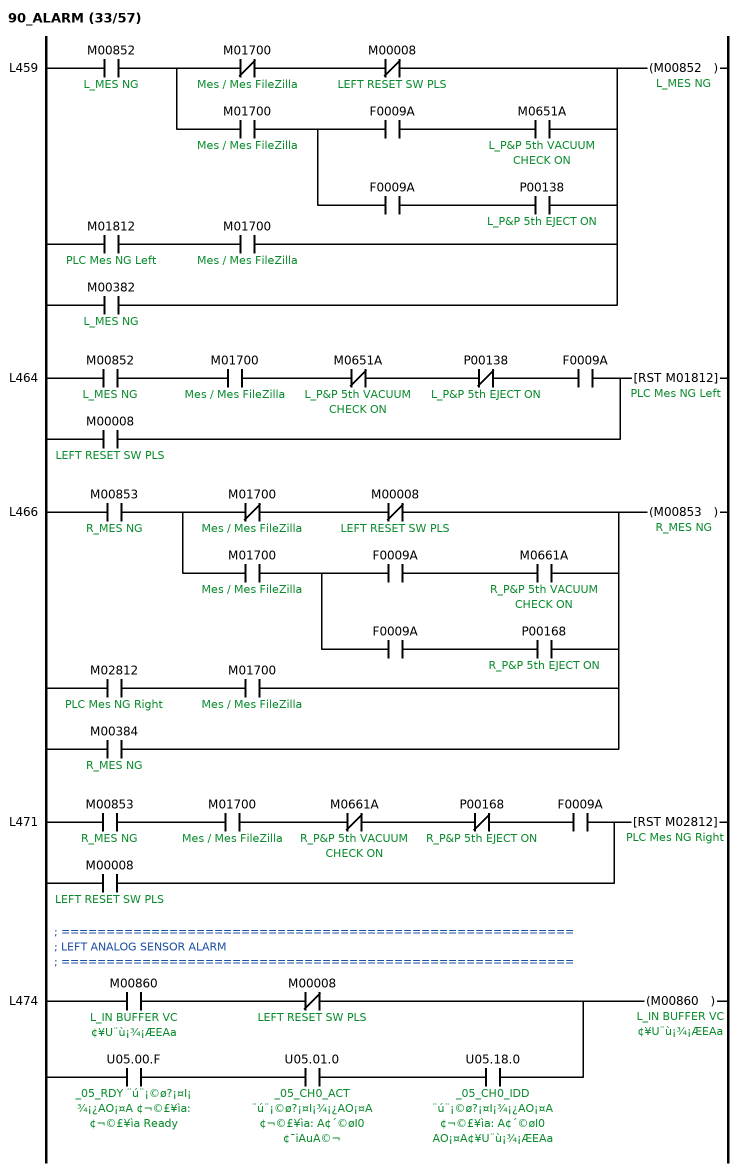
[picture p384: 90_ALARM rungs L459-L474]
; L459
LOAD      M00852	// L_MES NG
LOAD NOT  M01700	// Mes / Mes FileZilla
AND NOT   M00008	// LEFT RESET SW PLS
LOAD      M01700	// Mes / Mes FileZilla
LOAD      F0009A
AND       M0651A	// L_P&P 5th VACUUM CHECK ON
LOAD      F0009A
AND       P00138	// L_P&P 5th EJECT ON
OR LOAD
AND LOAD
OR LOAD
AND LOAD
LOAD      M01812	// PLC Mes NG Left
AND       M01700	// Mes / Mes FileZilla
OR LOAD
OR        M00382	// L_MES NG
OUT       M00852	// L_MES NG
; L464
LOAD      M00852	// L_MES NG
AND       M01700	// Mes / Mes FileZilla
AND NOT   M0651A	// L_P&P 5th VACUUM CHECK ON
AND NOT   P00138	// L_P&P 5th EJECT ON
AND       F0009A
OR        M00008	// LEFT RESET SW PLS
RST       M01812	// PLC Mes NG Left
; L466
LOAD      M00853	// R_MES NG
LOAD NOT  M01700	// Mes / Mes FileZilla
AND NOT   M00008	// LEFT RESET SW PLS
LOAD      M01700	// Mes / Mes FileZilla
LOAD      F0009A
AND       M0661A	// R_P&P 5th VACUUM CHECK ON
LOAD      F0009A
AND       P00168	// R_P&P 5th EJECT ON
OR LOAD
AND LOAD
OR LOAD
AND LOAD
LOAD      M02812	// PLC Mes NG Right
AND       M01700	// Mes / Mes FileZilla
OR LOAD
OR        M00384	// R_MES NG
OUT       M00853	// R_MES NG
; L471
LOAD      M00853	// R_MES NG
AND       M01700	// Mes / Mes FileZilla
AND NOT   M0661A	// R_P&P 5th VACUUM CHECK ON
AND NOT   P00168	// R_P&P 5th EJECT ON
AND       F0009A
OR        M00008	// LEFT RESET SW PLS
RST       M02812	// PLC Mes NG Right
// =========================================================
// 
//        LEFT ANALOG SENSOR ALARM
// 
// =========================================================
; L474
LOAD      M00860	// L_IN BUFFER VC ¢¥U¨ù¡¾¡ÆEAa
AND NOT   M00008	// LEFT RESET SW PLS
LOAD      U05.00.F	// _05_RDY ¨ú¨¡©ø?¡¤I¡¾¡¿AO¡¤A ¢¬©£¥ìa: ¢¬©£¥ìa Ready
AND       U05.01.0	// _05_CH0_ACT ¨ú¨¡©ø?¡¤I¡¾¡¿AO¡¤A ¢¬©£¥ìa: A¢´©øI0 ¢¯iAuA©¬
AND       U05.18.0	// _05_CH0_IDD ¨ú¨¡©ø?¡¤I¡¾¡¿AO¡¤A ¢¬©£¥ìa: A¢´©øI0 AO¡¤A¢¥U¨ù¡¾¡ÆEAa
OR LOAD
OUT       M00860	// L_IN BUFFER VC ¢¥U¨ù¡¾¡ÆEAa

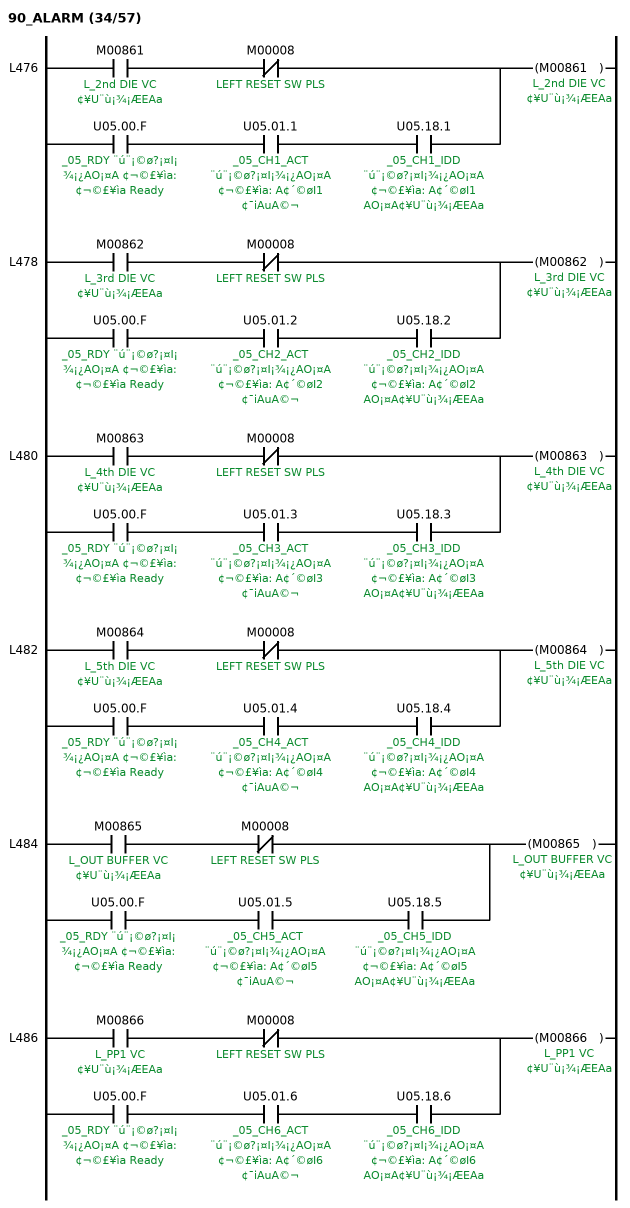
; L476
LOAD      M00861	// L_2nd DIE VC ¢¥U¨ù¡¾¡ÆEAa
AND NOT   M00008	// LEFT RESET SW PLS
LOAD      U05.00.F	// _05_RDY ¨ú¨¡©ø?¡¤I¡¾¡¿AO¡¤A ¢¬©£¥ìa: ¢¬©£¥ìa Ready
AND       U05.01.1	// _05_CH1_ACT ¨ú¨¡©ø?¡¤I¡¾¡¿AO¡¤A ¢¬©£¥ìa: A¢´©øI1 ¢¯iAuA©¬
AND       U05.18.1	// _05_CH1_IDD ¨ú¨¡©ø?¡¤I¡¾¡¿AO¡¤A ¢¬©£¥ìa: A¢´©øI1 AO¡¤A¢¥U¨ù¡¾¡ÆEAa
OR LOAD
OUT       M00861	// L_2nd DIE VC ¢¥U¨ù¡¾¡ÆEAa
; L478
LOAD      M00862	// L_3rd DIE VC ¢¥U¨ù¡¾¡ÆEAa
AND NOT   M00008	// LEFT RESET SW PLS
LOAD      U05.00.F	// _05_RDY ¨ú¨¡©ø?¡¤I¡¾¡¿AO¡¤A ¢¬©£¥ìa: ¢¬©£¥ìa Ready
AND       U05.01.2	// _05_CH2_ACT ¨ú¨¡©ø?¡¤I¡¾¡¿AO¡¤A ¢¬©£¥ìa: A¢´©øI2 ¢¯iAuA©¬
AND       U05.18.2	// _05_CH2_IDD ¨ú¨¡©ø?¡¤I¡¾¡¿AO¡¤A ¢¬©£¥ìa: A¢´©øI2 AO¡¤A¢¥U¨ù¡¾¡ÆEAa
OR LOAD
OUT       M00862	// L_3rd DIE VC ¢¥U¨ù¡¾¡ÆEAa
; L480
LOAD      M00863	// L_4th DIE VC ¢¥U¨ù¡¾¡ÆEAa
AND NOT   M00008	// LEFT RESET SW PLS
LOAD      U05.00.F	// _05_RDY ¨ú¨¡©ø?¡¤I¡¾¡¿AO¡¤A ¢¬©£¥ìa: ¢¬©£¥ìa Ready
AND       U05.01.3	// _05_CH3_ACT ¨ú¨¡©ø?¡¤I¡¾¡¿AO¡¤A ¢¬©£¥ìa: A¢´©øI3 ¢¯iAuA©¬
AND       U05.18.3	// _05_CH3_IDD ¨ú¨¡©ø?¡¤I¡¾¡¿AO¡¤A ¢¬©£¥ìa: A¢´©øI3 AO¡¤A¢¥U¨ù¡¾¡ÆEAa
OR LOAD
OUT       M00863	// L_4th DIE VC ¢¥U¨ù¡¾¡ÆEAa
; L482
LOAD      M00864	// L_5th DIE VC ¢¥U¨ù¡¾¡ÆEAa
AND NOT   M00008	// LEFT RESET SW PLS
LOAD      U05.00.F	// _05_RDY ¨ú¨¡©ø?¡¤I¡¾¡¿AO¡¤A ¢¬©£¥ìa: ¢¬©£¥ìa Ready
AND       U05.01.4	// _05_CH4_ACT ¨ú¨¡©ø?¡¤I¡¾¡¿AO¡¤A ¢¬©£¥ìa: A¢´©øI4 ¢¯iAuA©¬
AND       U05.18.4	// _05_CH4_IDD ¨ú¨¡©ø?¡¤I¡¾¡¿AO¡¤A ¢¬©£¥ìa: A¢´©øI4 AO¡¤A¢¥U¨ù¡¾¡ÆEAa
OR LOAD
OUT       M00864	// L_5th DIE VC ¢¥U¨ù¡¾¡ÆEAa
; L484
LOAD      M00865	// L_OUT BUFFER VC ¢¥U¨ù¡¾¡ÆEAa
AND NOT   M00008	// LEFT RESET SW PLS
LOAD      U05.00.F	// _05_RDY ¨ú¨¡©ø?¡¤I¡¾¡¿AO¡¤A ¢¬©£¥ìa: ¢¬©£¥ìa Ready
AND       U05.01.5	// _05_CH5_ACT ¨ú¨¡©ø?¡¤I¡¾¡¿AO¡¤A ¢¬©£¥ìa: A¢´©øI5 ¢¯iAuA©¬
AND       U05.18.5	// _05_CH5_IDD ¨ú¨¡©ø?¡¤I¡¾¡¿AO¡¤A ¢¬©£¥ìa: A¢´©øI5 AO¡¤A¢¥U¨ù¡¾¡ÆEAa
OR LOAD
OUT       M00865	// L_OUT BUFFER VC ¢¥U¨ù¡¾¡ÆEAa
; L486
LOAD      M00866	// L_PP1 VC ¢¥U¨ù¡¾¡ÆEAa
AND NOT   M00008	// LEFT RESET SW PLS
LOAD      U05.00.F	// _05_RDY ¨ú¨¡©ø?¡¤I¡¾¡¿AO¡¤A ¢¬©£¥ìa: ¢¬©£¥ìa Ready
AND       U05.01.6	// _05_CH6_ACT ¨ú¨¡©ø?¡¤I¡¾¡¿AO¡¤A ¢¬©£¥ìa: A¢´©øI6 ¢¯iAuA©¬
AND       U05.18.6	// _05_CH6_IDD ¨ú¨¡©ø?¡¤I¡¾¡¿AO¡¤A ¢¬©£¥ìa: A¢´©øI6 AO¡¤A¢¥U¨ù¡¾¡ÆEAa
OR LOAD
OUT       M00866	// L_PP1 VC ¢¥U¨ù¡¾¡ÆEAa

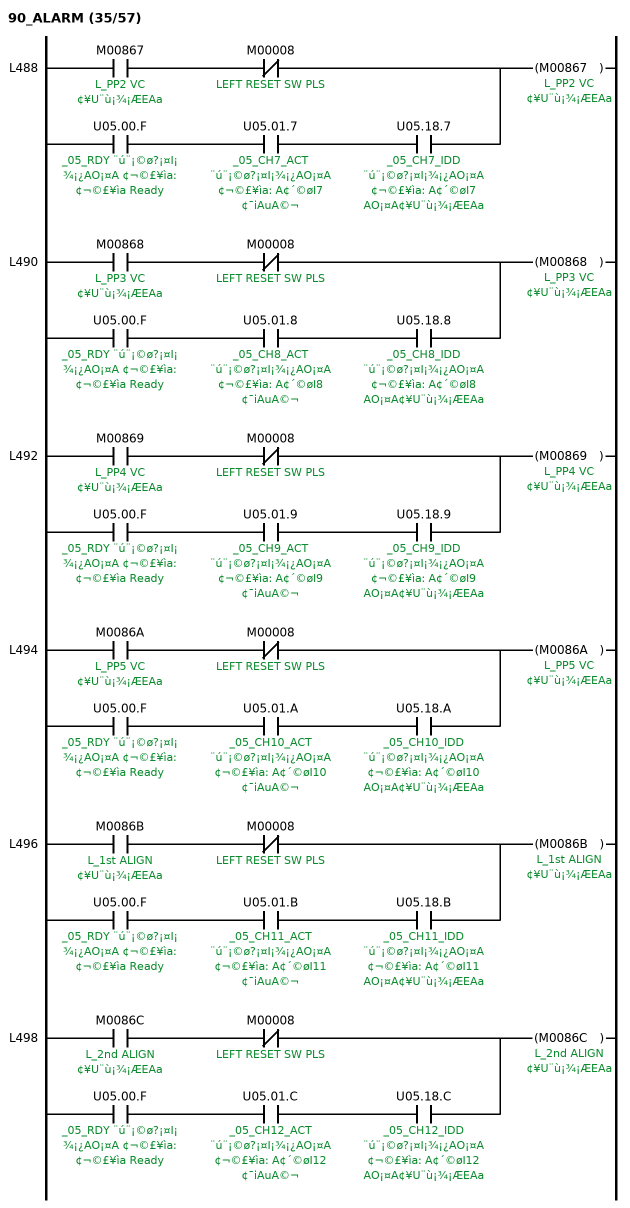
; L488
LOAD      M00867	// L_PP2 VC ¢¥U¨ù¡¾¡ÆEAa
AND NOT   M00008	// LEFT RESET SW PLS
LOAD      U05.00.F	// _05_RDY ¨ú¨¡©ø?¡¤I¡¾¡¿AO¡¤A ¢¬©£¥ìa: ¢¬©£¥ìa Ready
AND       U05.01.7	// _05_CH7_ACT ¨ú¨¡©ø?¡¤I¡¾¡¿AO¡¤A ¢¬©£¥ìa: A¢´©øI7 ¢¯iAuA©¬
AND       U05.18.7	// _05_CH7_IDD ¨ú¨¡©ø?¡¤I¡¾¡¿AO¡¤A ¢¬©£¥ìa: A¢´©øI7 AO¡¤A¢¥U¨ù¡¾¡ÆEAa
OR LOAD
OUT       M00867	// L_PP2 VC ¢¥U¨ù¡¾¡ÆEAa
; L490
LOAD      M00868	// L_PP3 VC ¢¥U¨ù¡¾¡ÆEAa
AND NOT   M00008	// LEFT RESET SW PLS
LOAD      U05.00.F	// _05_RDY ¨ú¨¡©ø?¡¤I¡¾¡¿AO¡¤A ¢¬©£¥ìa: ¢¬©£¥ìa Ready
AND       U05.01.8	// _05_CH8_ACT ¨ú¨¡©ø?¡¤I¡¾¡¿AO¡¤A ¢¬©£¥ìa: A¢´©øI8 ¢¯iAuA©¬
AND       U05.18.8	// _05_CH8_IDD ¨ú¨¡©ø?¡¤I¡¾¡¿AO¡¤A ¢¬©£¥ìa: A¢´©øI8 AO¡¤A¢¥U¨ù¡¾¡ÆEAa
OR LOAD
OUT       M00868	// L_PP3 VC ¢¥U¨ù¡¾¡ÆEAa
; L492
LOAD      M00869	// L_PP4 VC ¢¥U¨ù¡¾¡ÆEAa
AND NOT   M00008	// LEFT RESET SW PLS
LOAD      U05.00.F	// _05_RDY ¨ú¨¡©ø?¡¤I¡¾¡¿AO¡¤A ¢¬©£¥ìa: ¢¬©£¥ìa Ready
AND       U05.01.9	// _05_CH9_ACT ¨ú¨¡©ø?¡¤I¡¾¡¿AO¡¤A ¢¬©£¥ìa: A¢´©øI9 ¢¯iAuA©¬
AND       U05.18.9	// _05_CH9_IDD ¨ú¨¡©ø?¡¤I¡¾¡¿AO¡¤A ¢¬©£¥ìa: A¢´©øI9 AO¡¤A¢¥U¨ù¡¾¡ÆEAa
OR LOAD
OUT       M00869	// L_PP4 VC ¢¥U¨ù¡¾¡ÆEAa
; L494
LOAD      M0086A	// L_PP5 VC ¢¥U¨ù¡¾¡ÆEAa
AND NOT   M00008	// LEFT RESET SW PLS
LOAD      U05.00.F	// _05_RDY ¨ú¨¡©ø?¡¤I¡¾¡¿AO¡¤A ¢¬©£¥ìa: ¢¬©£¥ìa Ready
AND       U05.01.A	// _05_CH10_ACT ¨ú¨¡©ø?¡¤I¡¾¡¿AO¡¤A ¢¬©£¥ìa: A¢´©øI10 ¢¯iAuA©¬
AND       U05.18.A	// _05_CH10_IDD ¨ú¨¡©ø?¡¤I¡¾¡¿AO¡¤A ¢¬©£¥ìa: A¢´©øI10 AO¡¤A¢¥U¨ù¡¾¡ÆEAa
OR LOAD
OUT       M0086A	// L_PP5 VC ¢¥U¨ù¡¾¡ÆEAa
; L496
LOAD      M0086B	// L_1st ALIGN ¢¥U¨ù¡¾¡ÆEAa
AND NOT   M00008	// LEFT RESET SW PLS
LOAD      U05.00.F	// _05_RDY ¨ú¨¡©ø?¡¤I¡¾¡¿AO¡¤A ¢¬©£¥ìa: ¢¬©£¥ìa Ready
AND       U05.01.B	// _05_CH11_ACT ¨ú¨¡©ø?¡¤I¡¾¡¿AO¡¤A ¢¬©£¥ìa: A¢´©øI11 ¢¯iAuA©¬
AND       U05.18.B	// _05_CH11_IDD ¨ú¨¡©ø?¡¤I¡¾¡¿AO¡¤A ¢¬©£¥ìa: A¢´©øI11 AO¡¤A¢¥U¨ù¡¾¡ÆEAa
OR LOAD
OUT       M0086B	// L_1st ALIGN ¢¥U¨ù¡¾¡ÆEAa
; L498
LOAD      M0086C	// L_2nd ALIGN ¢¥U¨ù¡¾¡ÆEAa
AND NOT   M00008	// LEFT RESET SW PLS
LOAD      U05.00.F	// _05_RDY ¨ú¨¡©ø?¡¤I¡¾¡¿AO¡¤A ¢¬©£¥ìa: ¢¬©£¥ìa Ready
AND       U05.01.C	// _05_CH12_ACT ¨ú¨¡©ø?¡¤I¡¾¡¿AO¡¤A ¢¬©£¥ìa: A¢´©øI12 ¢¯iAuA©¬
AND       U05.18.C	// _05_CH12_IDD ¨ú¨¡©ø?¡¤I¡¾¡¿AO¡¤A ¢¬©£¥ìa: A¢´©øI12 AO¡¤A¢¥U¨ù¡¾¡ÆEAa
OR LOAD
OUT       M0086C	// L_2nd ALIGN ¢¥U¨ù¡¾¡ÆEAa

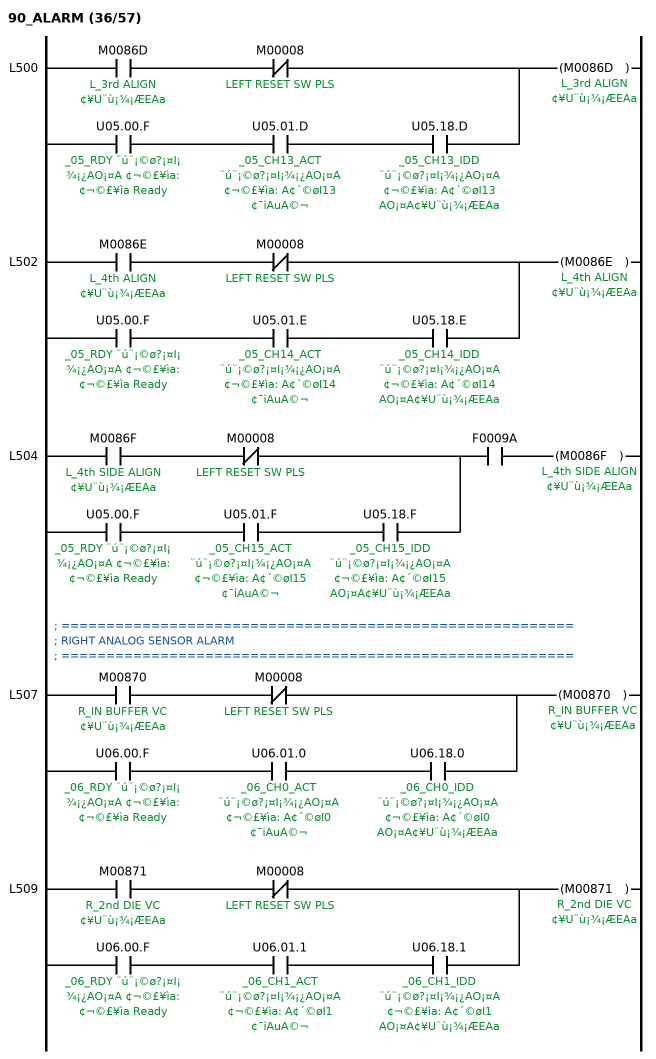
; L500
LOAD      M0086D	// L_3rd ALIGN ¢¥U¨ù¡¾¡ÆEAa
AND NOT   M00008	// LEFT RESET SW PLS
LOAD      U05.00.F	// _05_RDY ¨ú¨¡©ø?¡¤I¡¾¡¿AO¡¤A ¢¬©£¥ìa: ¢¬©£¥ìa Ready
AND       U05.01.D	// _05_CH13_ACT ¨ú¨¡©ø?¡¤I¡¾¡¿AO¡¤A ¢¬©£¥ìa: A¢´©øI13 ¢¯iAuA©¬
AND       U05.18.D	// _05_CH13_IDD ¨ú¨¡©ø?¡¤I¡¾¡¿AO¡¤A ¢¬©£¥ìa: A¢´©øI13 AO¡¤A¢¥U¨ù¡¾¡ÆEAa
OR LOAD
OUT       M0086D	// L_3rd ALIGN ¢¥U¨ù¡¾¡ÆEAa
; L502
LOAD      M0086E	// L_4th ALIGN ¢¥U¨ù¡¾¡ÆEAa
AND NOT   M00008	// LEFT RESET SW PLS
LOAD      U05.00.F	// _05_RDY ¨ú¨¡©ø?¡¤I¡¾¡¿AO¡¤A ¢¬©£¥ìa: ¢¬©£¥ìa Ready
AND       U05.01.E	// _05_CH14_ACT ¨ú¨¡©ø?¡¤I¡¾¡¿AO¡¤A ¢¬©£¥ìa: A¢´©øI14 ¢¯iAuA©¬
AND       U05.18.E	// _05_CH14_IDD ¨ú¨¡©ø?¡¤I¡¾¡¿AO¡¤A ¢¬©£¥ìa: A¢´©øI14 AO¡¤A¢¥U¨ù¡¾¡ÆEAa
OR LOAD
OUT       M0086E	// L_4th ALIGN ¢¥U¨ù¡¾¡ÆEAa
; L504
LOAD      M0086F	// L_4th SIDE ALIGN ¢¥U¨ù¡¾¡ÆEAa
AND NOT   M00008	// LEFT RESET SW PLS
LOAD      U05.00.F	// _05_RDY ¨ú¨¡©ø?¡¤I¡¾¡¿AO¡¤A ¢¬©£¥ìa: ¢¬©£¥ìa Ready
AND       U05.01.F	// _05_CH15_ACT ¨ú¨¡©ø?¡¤I¡¾¡¿AO¡¤A ¢¬©£¥ìa: A¢´©øI15 ¢¯iAuA©¬
AND       U05.18.F	// _05_CH15_IDD ¨ú¨¡©ø?¡¤I¡¾¡¿AO¡¤A ¢¬©£¥ìa: A¢´©øI15 AO¡¤A¢¥U¨ù¡¾¡ÆEAa
OR LOAD
AND       F0009A
OUT       M0086F	// L_4th SIDE ALIGN ¢¥U¨ù¡¾¡ÆEAa
// =========================================================
// 
//        RIGHT ANALOG SENSOR ALARM
// 
// =========================================================
; L507
LOAD      M00870	// R_IN BUFFER VC ¢¥U¨ù¡¾¡ÆEAa
AND NOT   M00008	// LEFT RESET SW PLS
LOAD      U06.00.F	// _06_RDY ¨ú¨¡©ø?¡¤I¡¾¡¿AO¡¤A ¢¬©£¥ìa: ¢¬©£¥ìa Ready
AND       U06.01.0	// _06_CH0_ACT ¨ú¨¡©ø?¡¤I¡¾¡¿AO¡¤A ¢¬©£¥ìa: A¢´©øI0 ¢¯iAuA©¬
AND       U06.18.0	// _06_CH0_IDD ¨ú¨¡©ø?¡¤I¡¾¡¿AO¡¤A ¢¬©£¥ìa: A¢´©øI0 AO¡¤A¢¥U¨ù¡¾¡ÆEAa
OR LOAD
OUT       M00870	// R_IN BUFFER VC ¢¥U¨ù¡¾¡ÆEAa
; L509
LOAD      M00871	// R_2nd DIE VC ¢¥U¨ù¡¾¡ÆEAa
AND NOT   M00008	// LEFT RESET SW PLS
LOAD      U06.00.F	// _06_RDY ¨ú¨¡©ø?¡¤I¡¾¡¿AO¡¤A ¢¬©£¥ìa: ¢¬©£¥ìa Ready
AND       U06.01.1	// _06_CH1_ACT ¨ú¨¡©ø?¡¤I¡¾¡¿AO¡¤A ¢¬©£¥ìa: A¢´©øI1 ¢¯iAuA©¬
AND       U06.18.1	// _06_CH1_IDD ¨ú¨¡©ø?¡¤I¡¾¡¿AO¡¤A ¢¬©£¥ìa: A¢´©øI1 AO¡¤A¢¥U¨ù¡¾¡ÆEAa
OR LOAD
OUT       M00871	// R_2nd DIE VC ¢¥U¨ù¡¾¡ÆEAa

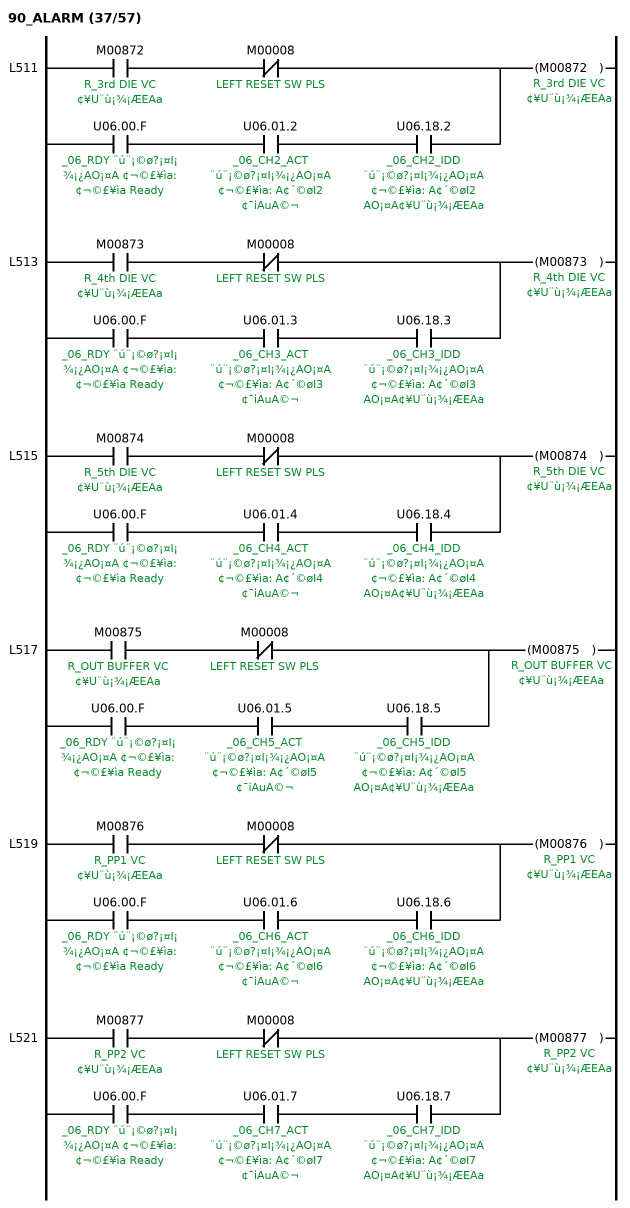
; L511
LOAD      M00872	// R_3rd DIE VC ¢¥U¨ù¡¾¡ÆEAa
AND NOT   M00008	// LEFT RESET SW PLS
LOAD      U06.00.F	// _06_RDY ¨ú¨¡©ø?¡¤I¡¾¡¿AO¡¤A ¢¬©£¥ìa: ¢¬©£¥ìa Ready
AND       U06.01.2	// _06_CH2_ACT ¨ú¨¡©ø?¡¤I¡¾¡¿AO¡¤A ¢¬©£¥ìa: A¢´©øI2 ¢¯iAuA©¬
AND       U06.18.2	// _06_CH2_IDD ¨ú¨¡©ø?¡¤I¡¾¡¿AO¡¤A ¢¬©£¥ìa: A¢´©øI2 AO¡¤A¢¥U¨ù¡¾¡ÆEAa
OR LOAD
OUT       M00872	// R_3rd DIE VC ¢¥U¨ù¡¾¡ÆEAa
; L513
LOAD      M00873	// R_4th DIE VC ¢¥U¨ù¡¾¡ÆEAa
AND NOT   M00008	// LEFT RESET SW PLS
LOAD      U06.00.F	// _06_RDY ¨ú¨¡©ø?¡¤I¡¾¡¿AO¡¤A ¢¬©£¥ìa: ¢¬©£¥ìa Ready
AND       U06.01.3	// _06_CH3_ACT ¨ú¨¡©ø?¡¤I¡¾¡¿AO¡¤A ¢¬©£¥ìa: A¢´©øI3 ¢¯iAuA©¬
AND       U06.18.3	// _06_CH3_IDD ¨ú¨¡©ø?¡¤I¡¾¡¿AO¡¤A ¢¬©£¥ìa: A¢´©øI3 AO¡¤A¢¥U¨ù¡¾¡ÆEAa
OR LOAD
OUT       M00873	// R_4th DIE VC ¢¥U¨ù¡¾¡ÆEAa
; L515
LOAD      M00874	// R_5th DIE VC ¢¥U¨ù¡¾¡ÆEAa
AND NOT   M00008	// LEFT RESET SW PLS
LOAD      U06.00.F	// _06_RDY ¨ú¨¡©ø?¡¤I¡¾¡¿AO¡¤A ¢¬©£¥ìa: ¢¬©£¥ìa Ready
AND       U06.01.4	// _06_CH4_ACT ¨ú¨¡©ø?¡¤I¡¾¡¿AO¡¤A ¢¬©£¥ìa: A¢´©øI4 ¢¯iAuA©¬
AND       U06.18.4	// _06_CH4_IDD ¨ú¨¡©ø?¡¤I¡¾¡¿AO¡¤A ¢¬©£¥ìa: A¢´©øI4 AO¡¤A¢¥U¨ù¡¾¡ÆEAa
OR LOAD
OUT       M00874	// R_5th DIE VC ¢¥U¨ù¡¾¡ÆEAa
; L517
LOAD      M00875	// R_OUT BUFFER VC ¢¥U¨ù¡¾¡ÆEAa
AND NOT   M00008	// LEFT RESET SW PLS
LOAD      U06.00.F	// _06_RDY ¨ú¨¡©ø?¡¤I¡¾¡¿AO¡¤A ¢¬©£¥ìa: ¢¬©£¥ìa Ready
AND       U06.01.5	// _06_CH5_ACT ¨ú¨¡©ø?¡¤I¡¾¡¿AO¡¤A ¢¬©£¥ìa: A¢´©øI5 ¢¯iAuA©¬
AND       U06.18.5	// _06_CH5_IDD ¨ú¨¡©ø?¡¤I¡¾¡¿AO¡¤A ¢¬©£¥ìa: A¢´©øI5 AO¡¤A¢¥U¨ù¡¾¡ÆEAa
OR LOAD
OUT       M00875	// R_OUT BUFFER VC ¢¥U¨ù¡¾¡ÆEAa
; L519
LOAD      M00876	// R_PP1 VC ¢¥U¨ù¡¾¡ÆEAa
AND NOT   M00008	// LEFT RESET SW PLS
LOAD      U06.00.F	// _06_RDY ¨ú¨¡©ø?¡¤I¡¾¡¿AO¡¤A ¢¬©£¥ìa: ¢¬©£¥ìa Ready
AND       U06.01.6	// _06_CH6_ACT ¨ú¨¡©ø?¡¤I¡¾¡¿AO¡¤A ¢¬©£¥ìa: A¢´©øI6 ¢¯iAuA©¬
AND       U06.18.6	// _06_CH6_IDD ¨ú¨¡©ø?¡¤I¡¾¡¿AO¡¤A ¢¬©£¥ìa: A¢´©øI6 AO¡¤A¢¥U¨ù¡¾¡ÆEAa
OR LOAD
OUT       M00876	// R_PP1 VC ¢¥U¨ù¡¾¡ÆEAa
; L521
LOAD      M00877	// R_PP2 VC ¢¥U¨ù¡¾¡ÆEAa
AND NOT   M00008	// LEFT RESET SW PLS
LOAD      U06.00.F	// _06_RDY ¨ú¨¡©ø?¡¤I¡¾¡¿AO¡¤A ¢¬©£¥ìa: ¢¬©£¥ìa Ready
AND       U06.01.7	// _06_CH7_ACT ¨ú¨¡©ø?¡¤I¡¾¡¿AO¡¤A ¢¬©£¥ìa: A¢´©øI7 ¢¯iAuA©¬
AND       U06.18.7	// _06_CH7_IDD ¨ú¨¡©ø?¡¤I¡¾¡¿AO¡¤A ¢¬©£¥ìa: A¢´©øI7 AO¡¤A¢¥U¨ù¡¾¡ÆEAa
OR LOAD
OUT       M00877	// R_PP2 VC ¢¥U¨ù¡¾¡ÆEAa

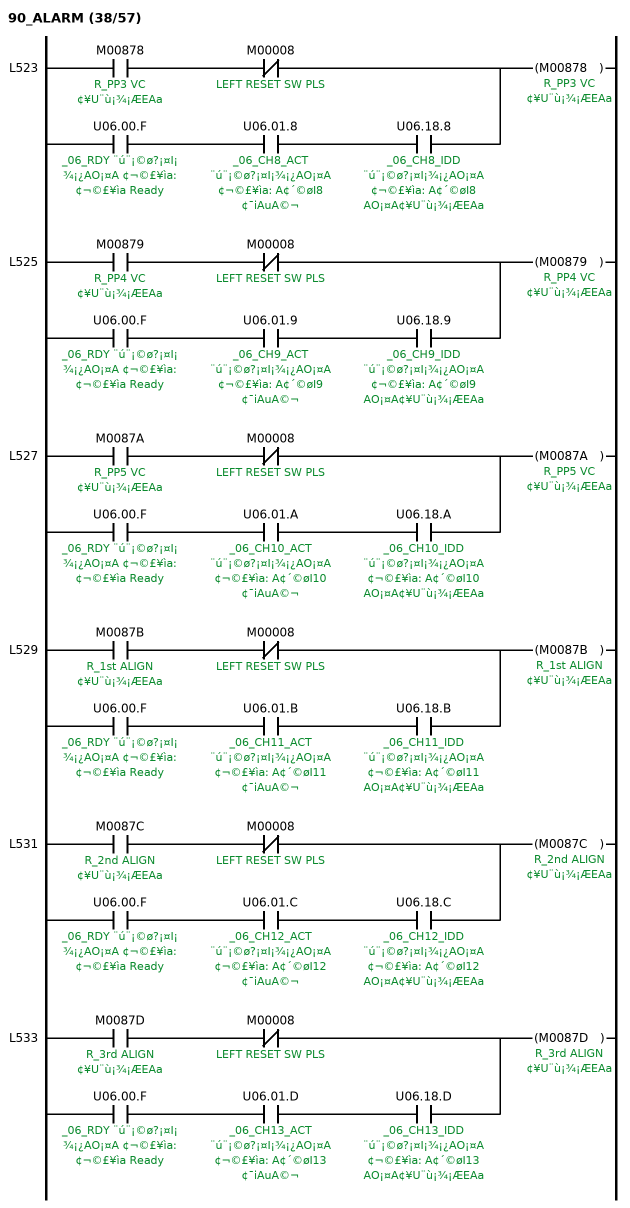
; L523
LOAD      M00878	// R_PP3 VC ¢¥U¨ù¡¾¡ÆEAa
AND NOT   M00008	// LEFT RESET SW PLS
LOAD      U06.00.F	// _06_RDY ¨ú¨¡©ø?¡¤I¡¾¡¿AO¡¤A ¢¬©£¥ìa: ¢¬©£¥ìa Ready
AND       U06.01.8	// _06_CH8_ACT ¨ú¨¡©ø?¡¤I¡¾¡¿AO¡¤A ¢¬©£¥ìa: A¢´©øI8 ¢¯iAuA©¬
AND       U06.18.8	// _06_CH8_IDD ¨ú¨¡©ø?¡¤I¡¾¡¿AO¡¤A ¢¬©£¥ìa: A¢´©øI8 AO¡¤A¢¥U¨ù¡¾¡ÆEAa
OR LOAD
OUT       M00878	// R_PP3 VC ¢¥U¨ù¡¾¡ÆEAa
; L525
LOAD      M00879	// R_PP4 VC ¢¥U¨ù¡¾¡ÆEAa
AND NOT   M00008	// LEFT RESET SW PLS
LOAD      U06.00.F	// _06_RDY ¨ú¨¡©ø?¡¤I¡¾¡¿AO¡¤A ¢¬©£¥ìa: ¢¬©£¥ìa Ready
AND       U06.01.9	// _06_CH9_ACT ¨ú¨¡©ø?¡¤I¡¾¡¿AO¡¤A ¢¬©£¥ìa: A¢´©øI9 ¢¯iAuA©¬
AND       U06.18.9	// _06_CH9_IDD ¨ú¨¡©ø?¡¤I¡¾¡¿AO¡¤A ¢¬©£¥ìa: A¢´©øI9 AO¡¤A¢¥U¨ù¡¾¡ÆEAa
OR LOAD
OUT       M00879	// R_PP4 VC ¢¥U¨ù¡¾¡ÆEAa
; L527
LOAD      M0087A	// R_PP5 VC ¢¥U¨ù¡¾¡ÆEAa
AND NOT   M00008	// LEFT RESET SW PLS
LOAD      U06.00.F	// _06_RDY ¨ú¨¡©ø?¡¤I¡¾¡¿AO¡¤A ¢¬©£¥ìa: ¢¬©£¥ìa Ready
AND       U06.01.A	// _06_CH10_ACT ¨ú¨¡©ø?¡¤I¡¾¡¿AO¡¤A ¢¬©£¥ìa: A¢´©øI10 ¢¯iAuA©¬
AND       U06.18.A	// _06_CH10_IDD ¨ú¨¡©ø?¡¤I¡¾¡¿AO¡¤A ¢¬©£¥ìa: A¢´©øI10 AO¡¤A¢¥U¨ù¡¾¡ÆEAa
OR LOAD
OUT       M0087A	// R_PP5 VC ¢¥U¨ù¡¾¡ÆEAa
; L529
LOAD      M0087B	// R_1st ALIGN ¢¥U¨ù¡¾¡ÆEAa
AND NOT   M00008	// LEFT RESET SW PLS
LOAD      U06.00.F	// _06_RDY ¨ú¨¡©ø?¡¤I¡¾¡¿AO¡¤A ¢¬©£¥ìa: ¢¬©£¥ìa Ready
AND       U06.01.B	// _06_CH11_ACT ¨ú¨¡©ø?¡¤I¡¾¡¿AO¡¤A ¢¬©£¥ìa: A¢´©øI11 ¢¯iAuA©¬
AND       U06.18.B	// _06_CH11_IDD ¨ú¨¡©ø?¡¤I¡¾¡¿AO¡¤A ¢¬©£¥ìa: A¢´©øI11 AO¡¤A¢¥U¨ù¡¾¡ÆEAa
OR LOAD
OUT       M0087B	// R_1st ALIGN ¢¥U¨ù¡¾¡ÆEAa
; L531
LOAD      M0087C	// R_2nd ALIGN ¢¥U¨ù¡¾¡ÆEAa
AND NOT   M00008	// LEFT RESET SW PLS
LOAD      U06.00.F	// _06_RDY ¨ú¨¡©ø?¡¤I¡¾¡¿AO¡¤A ¢¬©£¥ìa: ¢¬©£¥ìa Ready
AND       U06.01.C	// _06_CH12_ACT ¨ú¨¡©ø?¡¤I¡¾¡¿AO¡¤A ¢¬©£¥ìa: A¢´©øI12 ¢¯iAuA©¬
AND       U06.18.C	// _06_CH12_IDD ¨ú¨¡©ø?¡¤I¡¾¡¿AO¡¤A ¢¬©£¥ìa: A¢´©øI12 AO¡¤A¢¥U¨ù¡¾¡ÆEAa
OR LOAD
OUT       M0087C	// R_2nd ALIGN ¢¥U¨ù¡¾¡ÆEAa
; L533
LOAD      M0087D	// R_3rd ALIGN ¢¥U¨ù¡¾¡ÆEAa
AND NOT   M00008	// LEFT RESET SW PLS
LOAD      U06.00.F	// _06_RDY ¨ú¨¡©ø?¡¤I¡¾¡¿AO¡¤A ¢¬©£¥ìa: ¢¬©£¥ìa Ready
AND       U06.01.D	// _06_CH13_ACT ¨ú¨¡©ø?¡¤I¡¾¡¿AO¡¤A ¢¬©£¥ìa: A¢´©øI13 ¢¯iAuA©¬
AND       U06.18.D	// _06_CH13_IDD ¨ú¨¡©ø?¡¤I¡¾¡¿AO¡¤A ¢¬©£¥ìa: A¢´©øI13 AO¡¤A¢¥U¨ù¡¾¡ÆEAa
OR LOAD
OUT       M0087D	// R_3rd ALIGN ¢¥U¨ù¡¾¡ÆEAa

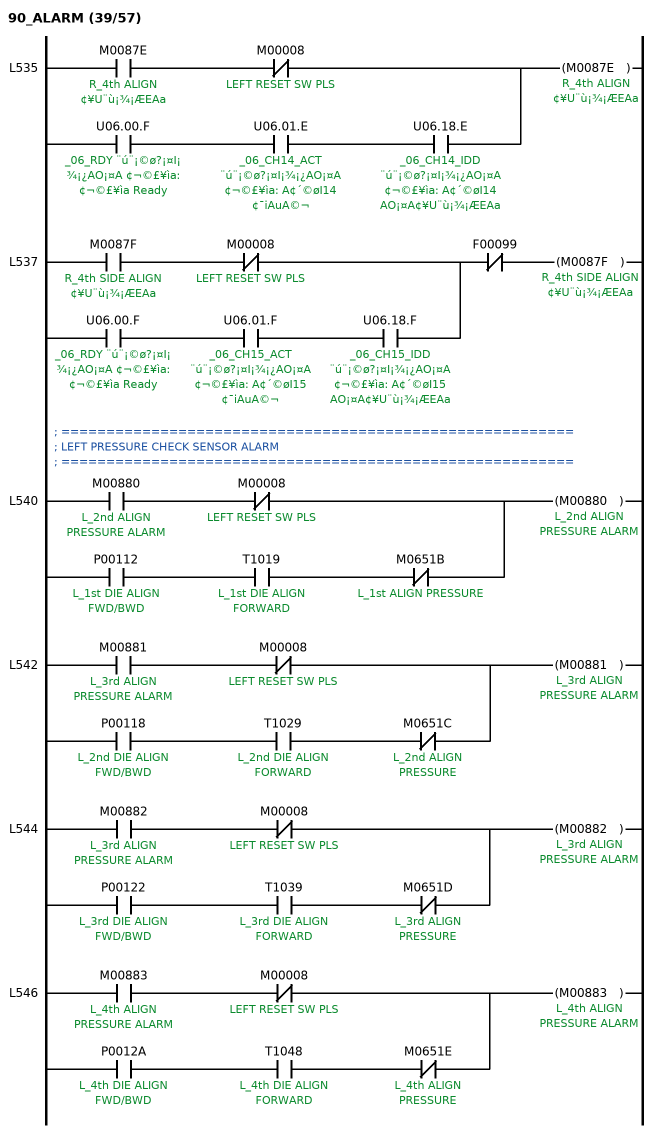
; L535
LOAD      M0087E	// R_4th ALIGN ¢¥U¨ù¡¾¡ÆEAa
AND NOT   M00008	// LEFT RESET SW PLS
LOAD      U06.00.F	// _06_RDY ¨ú¨¡©ø?¡¤I¡¾¡¿AO¡¤A ¢¬©£¥ìa: ¢¬©£¥ìa Ready
AND       U06.01.E	// _06_CH14_ACT ¨ú¨¡©ø?¡¤I¡¾¡¿AO¡¤A ¢¬©£¥ìa: A¢´©øI14 ¢¯iAuA©¬
AND       U06.18.E	// _06_CH14_IDD ¨ú¨¡©ø?¡¤I¡¾¡¿AO¡¤A ¢¬©£¥ìa: A¢´©øI14 AO¡¤A¢¥U¨ù¡¾¡ÆEAa
OR LOAD
OUT       M0087E	// R_4th ALIGN ¢¥U¨ù¡¾¡ÆEAa
; L537
LOAD      M0087F	// R_4th SIDE ALIGN ¢¥U¨ù¡¾¡ÆEAa
AND NOT   M00008	// LEFT RESET SW PLS
LOAD      U06.00.F	// _06_RDY ¨ú¨¡©ø?¡¤I¡¾¡¿AO¡¤A ¢¬©£¥ìa: ¢¬©£¥ìa Ready
AND       U06.01.F	// _06_CH15_ACT ¨ú¨¡©ø?¡¤I¡¾¡¿AO¡¤A ¢¬©£¥ìa: A¢´©øI15 ¢¯iAuA©¬
AND       U06.18.F	// _06_CH15_IDD ¨ú¨¡©ø?¡¤I¡¾¡¿AO¡¤A ¢¬©£¥ìa: A¢´©øI15 AO¡¤A¢¥U¨ù¡¾¡ÆEAa
OR LOAD
AND NOT   F00099
OUT       M0087F	// R_4th SIDE ALIGN ¢¥U¨ù¡¾¡ÆEAa
// =========================================================
// 
//        LEFT PRESSURE CHECK SENSOR ALARM
// 
// =========================================================
; L540
LOAD      M00880	// L_2nd ALIGN PRESSURE ALARM
AND NOT   M00008	// LEFT RESET SW PLS
LOAD      P00112	// L_1st DIE ALIGN FWD/BWD
AND       T1019	// L_1st DIE ALIGN FORWARD
AND NOT   M0651B	// L_1st ALIGN PRESSURE
OR LOAD
OUT       M00880	// L_2nd ALIGN PRESSURE ALARM
; L542
LOAD      M00881	// L_3rd ALIGN PRESSURE ALARM
AND NOT   M00008	// LEFT RESET SW PLS
LOAD      P00118	// L_2nd DIE ALIGN FWD/BWD
AND       T1029	// L_2nd DIE ALIGN FORWARD
AND NOT   M0651C	// L_2nd ALIGN PRESSURE
OR LOAD
OUT       M00881	// L_3rd ALIGN PRESSURE ALARM
; L544
LOAD      M00882	// L_3rd ALIGN PRESSURE ALARM
AND NOT   M00008	// LEFT RESET SW PLS
LOAD      P00122	// L_3rd DIE ALIGN FWD/BWD
AND       T1039	// L_3rd DIE ALIGN FORWARD
AND NOT   M0651D	// L_3rd ALIGN PRESSURE
OR LOAD
OUT       M00882	// L_3rd ALIGN PRESSURE ALARM
; L546
LOAD      M00883	// L_4th ALIGN PRESSURE ALARM
AND NOT   M00008	// LEFT RESET SW PLS
LOAD      P0012A	// L_4th DIE ALIGN FWD/BWD
AND       T1048	// L_4th DIE ALIGN FORWARD
AND NOT   M0651E	// L_4th ALIGN PRESSURE
OR LOAD
OUT       M00883	// L_4th ALIGN PRESSURE ALARM

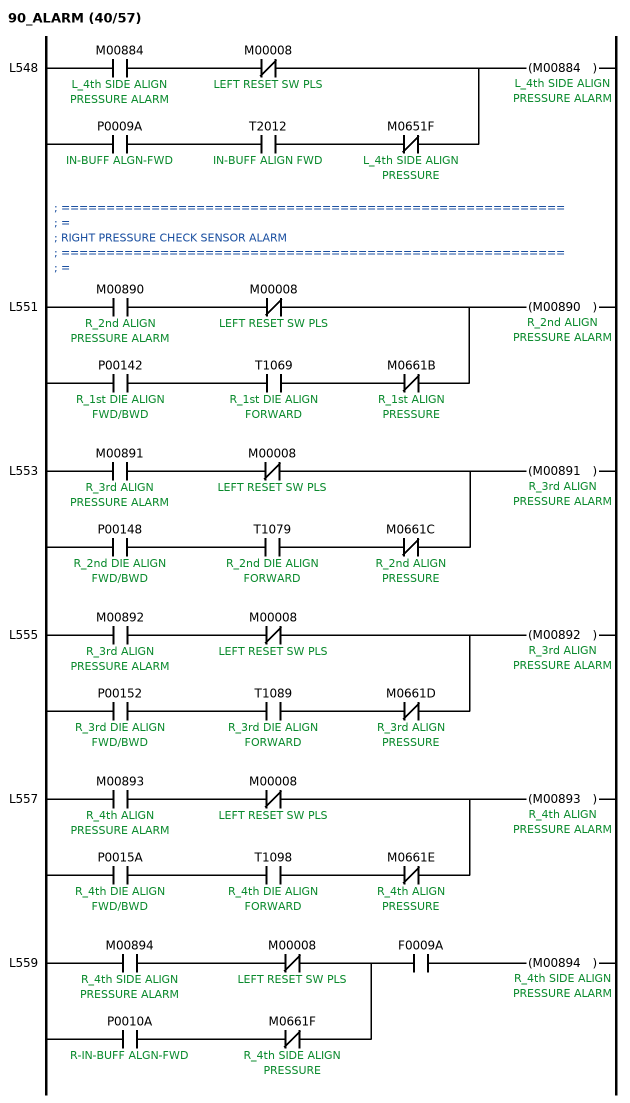
; L548
LOAD      M00884	// L_4th SIDE ALIGN PRESSURE ALARM
AND NOT   M00008	// LEFT RESET SW PLS
LOAD      P0009A	// IN-BUFF ALGN-FWD
AND       T2012	// IN-BUFF ALIGN FWD
AND NOT   M0651F	// L_4th SIDE ALIGN PRESSURE
OR LOAD
OUT       M00884	// L_4th SIDE ALIGN PRESSURE ALARM
// =========================================================
// 
//        RIGHT PRESSURE CHECK SENSOR ALARM
// 
// =========================================================
; L551
LOAD      M00890	// R_2nd ALIGN PRESSURE ALARM
AND NOT   M00008	// LEFT RESET SW PLS
LOAD      P00142	// R_1st DIE ALIGN FWD/BWD
AND       T1069	// R_1st DIE ALIGN FORWARD
AND NOT   M0661B	// R_1st ALIGN PRESSURE
OR LOAD
OUT       M00890	// R_2nd ALIGN PRESSURE ALARM
; L553
LOAD      M00891	// R_3rd ALIGN PRESSURE ALARM
AND NOT   M00008	// LEFT RESET SW PLS
LOAD      P00148	// R_2nd DIE ALIGN FWD/BWD
AND       T1079	// R_2nd DIE ALIGN FORWARD
AND NOT   M0661C	// R_2nd ALIGN PRESSURE
OR LOAD
OUT       M00891	// R_3rd ALIGN PRESSURE ALARM
; L555
LOAD      M00892	// R_3rd ALIGN PRESSURE ALARM
AND NOT   M00008	// LEFT RESET SW PLS
LOAD      P00152	// R_3rd DIE ALIGN FWD/BWD
AND       T1089	// R_3rd DIE ALIGN FORWARD
AND NOT   M0661D	// R_3rd ALIGN PRESSURE
OR LOAD
OUT       M00892	// R_3rd ALIGN PRESSURE ALARM
; L557
LOAD      M00893	// R_4th ALIGN PRESSURE ALARM
AND NOT   M00008	// LEFT RESET SW PLS
LOAD      P0015A	// R_4th DIE ALIGN FWD/BWD
AND       T1098	// R_4th DIE ALIGN FORWARD
AND NOT   M0661E	// R_4th ALIGN PRESSURE
OR LOAD
OUT       M00893	// R_4th ALIGN PRESSURE ALARM
; L559
LOAD      M00894	// R_4th SIDE ALIGN PRESSURE ALARM
AND NOT   M00008	// LEFT RESET SW PLS
LOAD      P0010A	// R-IN-BUFF ALGN-FWD
AND NOT   M0661F	// R_4th SIDE ALIGN PRESSURE
OR LOAD
AND       F0009A
OUT       M00894	// R_4th SIDE ALIGN PRESSURE ALARM

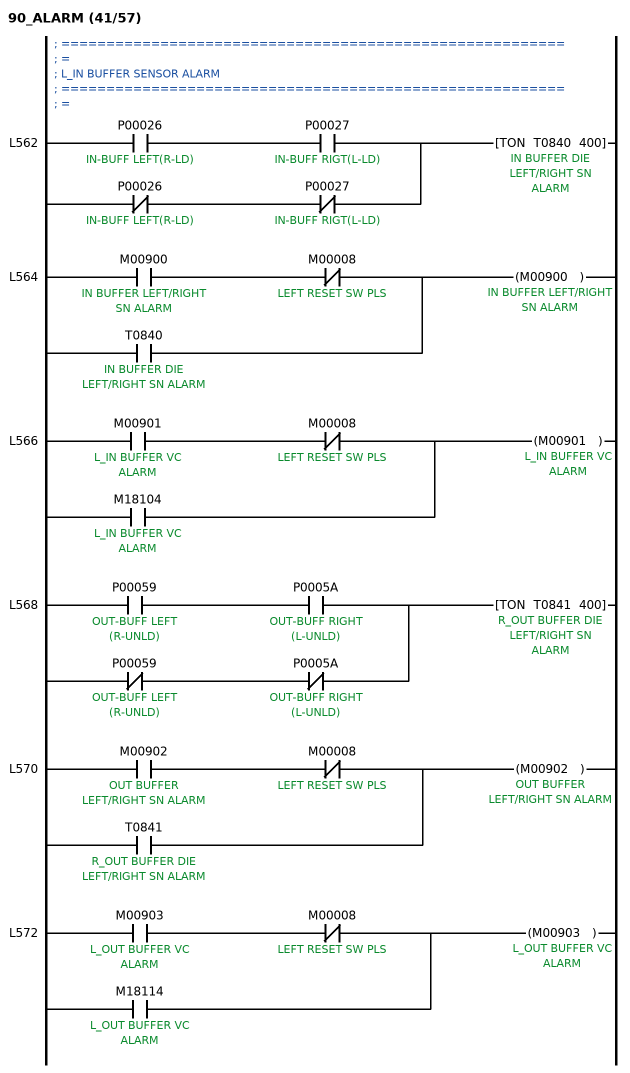
// =========================================================
// 
//        L_IN BUFFER SENSOR ALARM
// 
// =========================================================
; L562
LOAD      P00026	// IN-BUFF LEFT(R-LD)
AND       P00027	// IN-BUFF RIGT(L-LD)
LOAD NOT  P00026	// IN-BUFF LEFT(R-LD)
AND NOT   P00027	// IN-BUFF RIGT(L-LD)
OR LOAD
TON       T0840 400	// IN BUFFER DIE LEFT/RIGHT SN ALARM
; L564
LOAD      M00900	// IN BUFFER LEFT/RIGHT SN ALARM
AND NOT   M00008	// LEFT RESET SW PLS
OR        T0840	// IN BUFFER DIE LEFT/RIGHT SN ALARM
OUT       M00900	// IN BUFFER LEFT/RIGHT SN ALARM
; L566
LOAD      M00901	// L_IN BUFFER VC ALARM
AND NOT   M00008	// LEFT RESET SW PLS
OR        M18104	// L_IN BUFFER VC ALARM
OUT       M00901	// L_IN BUFFER VC ALARM
; L568
LOAD      P00059	// OUT-BUFF LEFT (R-UNLD)
AND       P0005A	// OUT-BUFF RIGHT (L-UNLD)
LOAD NOT  P00059	// OUT-BUFF LEFT (R-UNLD)
AND NOT   P0005A	// OUT-BUFF RIGHT (L-UNLD)
OR LOAD
TON       T0841 400	// R_OUT BUFFER DIE LEFT/RIGHT SN ALARM
; L570
LOAD      M00902	// OUT BUFFER LEFT/RIGHT SN ALARM
AND NOT   M00008	// LEFT RESET SW PLS
OR        T0841	// R_OUT BUFFER DIE LEFT/RIGHT SN ALARM
OUT       M00902	// OUT BUFFER LEFT/RIGHT SN ALARM
; L572
LOAD      M00903	// L_OUT BUFFER VC ALARM
AND NOT   M00008	// LEFT RESET SW PLS
OR        M18114	// L_OUT BUFFER VC ALARM
OUT       M00903	// L_OUT BUFFER VC ALARM

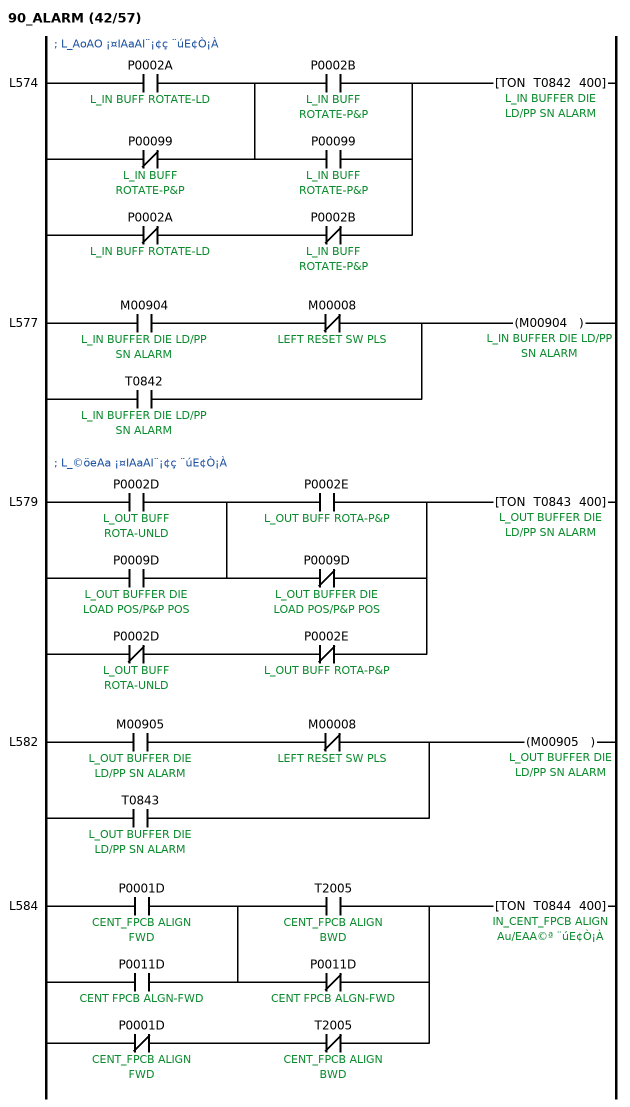
; L574
LOAD      P0002A	// L_IN BUFF ROTATE-LD
OR NOT    P00099	// L_IN BUFF ROTATE-P&P
LOAD      P0002B	// L_IN BUFF ROTATE-P&P
OR        P00099	// L_IN BUFF ROTATE-P&P
AND LOAD
LOAD NOT  P0002A	// L_IN BUFF ROTATE-LD
AND NOT   P0002B	// L_IN BUFF ROTATE-P&P
OR LOAD
TON       T0842 400	// L_IN BUFFER DIE LD/PP SN ALARM
// output comment: L_AoAO ¡¤IAaAI¨¡¢ç ¨úE¢Ò¡À
; L577
LOAD      M00904	// L_IN BUFFER DIE LD/PP SN ALARM
AND NOT   M00008	// LEFT RESET SW PLS
OR        T0842	// L_IN BUFFER DIE LD/PP SN ALARM
OUT       M00904	// L_IN BUFFER DIE LD/PP SN ALARM
; L579
LOAD      P0002D	// L_OUT BUFF ROTA-UNLD
OR        P0009D	// L_OUT BUFFER DIE LOAD POS/P&P POS
LOAD      P0002E	// L_OUT BUFF ROTA-P&P
OR NOT    P0009D	// L_OUT BUFFER DIE LOAD POS/P&P POS
AND LOAD
LOAD NOT  P0002D	// L_OUT BUFF ROTA-UNLD
AND NOT   P0002E	// L_OUT BUFF ROTA-P&P
OR LOAD
TON       T0843 400	// L_OUT BUFFER DIE LD/PP SN ALARM
// output comment: L_©öeAa ¡¤IAaAI¨¡¢ç ¨úE¢Ò¡À
; L582
LOAD      M00905	// L_OUT BUFFER DIE LD/PP SN ALARM
AND NOT   M00008	// LEFT RESET SW PLS
OR        T0843	// L_OUT BUFFER DIE LD/PP SN ALARM
OUT       M00905	// L_OUT BUFFER DIE LD/PP SN ALARM
; L584
LOAD      P0001D	// CENT_FPCB ALIGN FWD
OR        P0011D	// CENT FPCB ALGN-FWD
LOAD      T2005	// CENT_FPCB ALIGN BWD
OR NOT    P0011D	// CENT FPCB ALGN-FWD
AND LOAD
LOAD NOT  P0001D	// CENT_FPCB ALIGN FWD
AND NOT   T2005	// CENT_FPCB ALIGN BWD
OR LOAD
TON       T0844 400	// IN_CENT_FPCB ALIGN Au/EAA©ª ¨úE¢Ò¡À

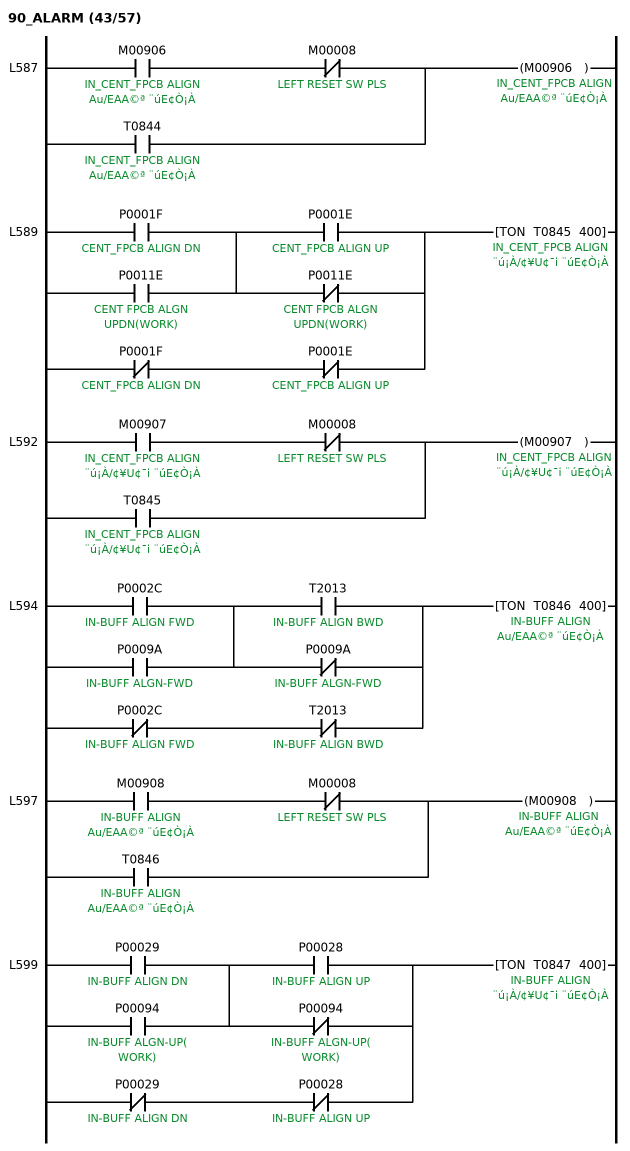
; L587
LOAD      M00906	// IN_CENT_FPCB ALIGN Au/EAA©ª ¨úE¢Ò¡À
AND NOT   M00008	// LEFT RESET SW PLS
OR        T0844	// IN_CENT_FPCB ALIGN Au/EAA©ª ¨úE¢Ò¡À
OUT       M00906	// IN_CENT_FPCB ALIGN Au/EAA©ª ¨úE¢Ò¡À
; L589
LOAD      P0001F	// CENT_FPCB ALIGN DN
OR        P0011E	// CENT FPCB ALGN UPDN(WORK)
LOAD      P0001E	// CENT_FPCB ALIGN UP
OR NOT    P0011E	// CENT FPCB ALGN UPDN(WORK)
AND LOAD
LOAD NOT  P0001F	// CENT_FPCB ALIGN DN
AND NOT   P0001E	// CENT_FPCB ALIGN UP
OR LOAD
TON       T0845 400	// IN_CENT_FPCB ALIGN ¨ú¡À/¢¥U¢¯i ¨úE¢Ò¡À
; L592
LOAD      M00907	// IN_CENT_FPCB ALIGN ¨ú¡À/¢¥U¢¯i ¨úE¢Ò¡À
AND NOT   M00008	// LEFT RESET SW PLS
OR        T0845	// IN_CENT_FPCB ALIGN ¨ú¡À/¢¥U¢¯i ¨úE¢Ò¡À
OUT       M00907	// IN_CENT_FPCB ALIGN ¨ú¡À/¢¥U¢¯i ¨úE¢Ò¡À
; L594
LOAD      P0002C	// IN-BUFF ALIGN FWD
OR        P0009A	// IN-BUFF ALGN-FWD
LOAD      T2013	// IN-BUFF ALIGN BWD
OR NOT    P0009A	// IN-BUFF ALGN-FWD
AND LOAD
LOAD NOT  P0002C	// IN-BUFF ALIGN FWD
AND NOT   T2013	// IN-BUFF ALIGN BWD
OR LOAD
TON       T0846 400	// IN-BUFF ALIGN Au/EAA©ª ¨úE¢Ò¡À
; L597
LOAD      M00908	// IN-BUFF ALIGN Au/EAA©ª ¨úE¢Ò¡À
AND NOT   M00008	// LEFT RESET SW PLS
OR        T0846	// IN-BUFF ALIGN Au/EAA©ª ¨úE¢Ò¡À
OUT       M00908	// IN-BUFF ALIGN Au/EAA©ª ¨úE¢Ò¡À
; L599
LOAD      P00029	// IN-BUFF ALIGN DN
OR        P00094	// IN-BUFF ALGN-UP(WORK)
LOAD      P00028	// IN-BUFF ALIGN UP
OR NOT    P00094	// IN-BUFF ALGN-UP(WORK)
AND LOAD
LOAD NOT  P00029	// IN-BUFF ALIGN DN
AND NOT   P00028	// IN-BUFF ALIGN UP
OR LOAD
TON       T0847 400	// IN-BUFF ALIGN ¨ú¡À/¢¥U¢¯i ¨úE¢Ò¡À

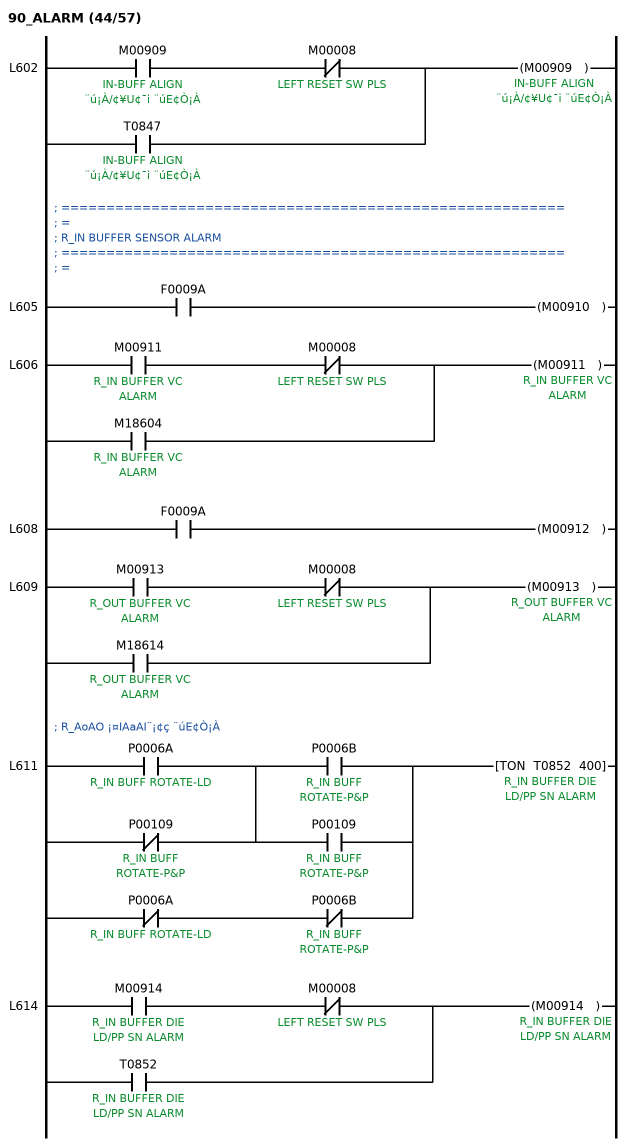
; L602
LOAD      M00909	// IN-BUFF ALIGN ¨ú¡À/¢¥U¢¯i ¨úE¢Ò¡À
AND NOT   M00008	// LEFT RESET SW PLS
OR        T0847	// IN-BUFF ALIGN ¨ú¡À/¢¥U¢¯i ¨úE¢Ò¡À
OUT       M00909	// IN-BUFF ALIGN ¨ú¡À/¢¥U¢¯i ¨úE¢Ò¡À
// =========================================================
// 
//        R_IN BUFFER SENSOR ALARM
// 
// =========================================================
; L605
LOAD      F0009A
OUT       M00910
; L606
LOAD      M00911	// R_IN BUFFER VC ALARM
AND NOT   M00008	// LEFT RESET SW PLS
OR        M18604	// R_IN BUFFER VC ALARM
OUT       M00911	// R_IN BUFFER VC ALARM
; L608
LOAD      F0009A
OUT       M00912
; L609
LOAD      M00913	// R_OUT BUFFER VC ALARM
AND NOT   M00008	// LEFT RESET SW PLS
OR        M18614	// R_OUT BUFFER VC ALARM
OUT       M00913	// R_OUT BUFFER VC ALARM
; L611
LOAD      P0006A	// R_IN BUFF ROTATE-LD
OR NOT    P00109	// R_IN BUFF ROTATE-P&P
LOAD      P0006B	// R_IN BUFF ROTATE-P&P
OR        P00109	// R_IN BUFF ROTATE-P&P
AND LOAD
LOAD NOT  P0006A	// R_IN BUFF ROTATE-LD
AND NOT   P0006B	// R_IN BUFF ROTATE-P&P
OR LOAD
TON       T0852 400	// R_IN BUFFER DIE LD/PP SN ALARM
// output comment: R_AoAO ¡¤IAaAI¨¡¢ç ¨úE¢Ò¡À
; L614
LOAD      M00914	// R_IN BUFFER DIE LD/PP SN ALARM
AND NOT   M00008	// LEFT RESET SW PLS
OR        T0852	// R_IN BUFFER DIE LD/PP SN ALARM
OUT       M00914	// R_IN BUFFER DIE LD/PP SN ALARM

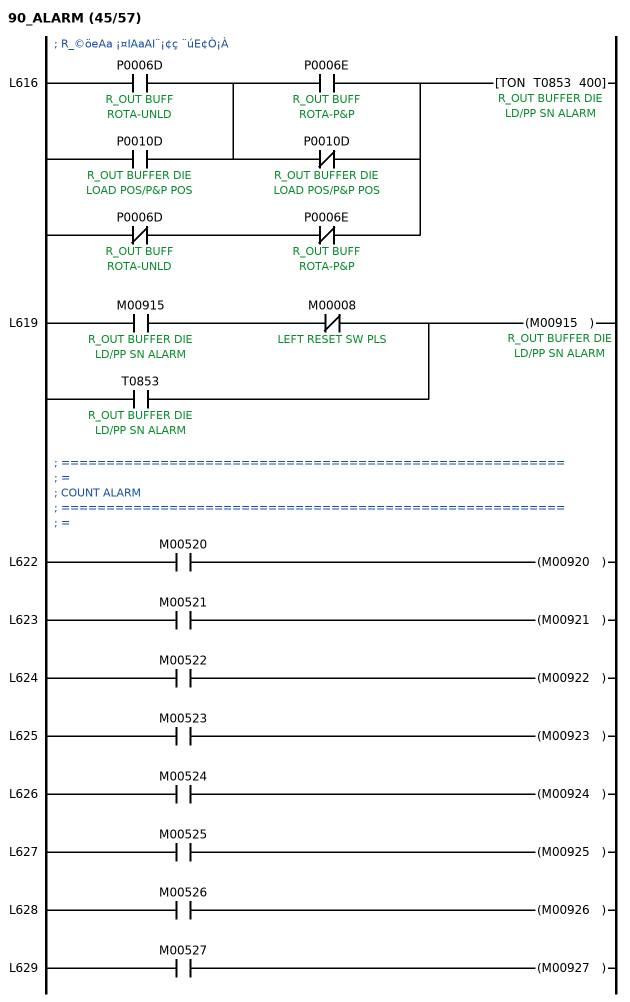
; L616
LOAD      P0006D	// R_OUT BUFF ROTA-UNLD
OR        P0010D	// R_OUT BUFFER DIE LOAD POS/P&P POS
LOAD      P0006E	// R_OUT BUFF ROTA-P&P
OR NOT    P0010D	// R_OUT BUFFER DIE LOAD POS/P&P POS
AND LOAD
LOAD NOT  P0006D	// R_OUT BUFF ROTA-UNLD
AND NOT   P0006E	// R_OUT BUFF ROTA-P&P
OR LOAD
TON       T0853 400	// R_OUT BUFFER DIE LD/PP SN ALARM
// output comment: R_©öeAa ¡¤IAaAI¨¡¢ç ¨úE¢Ò¡À
; L619
LOAD      M00915	// R_OUT BUFFER DIE LD/PP SN ALARM
AND NOT   M00008	// LEFT RESET SW PLS
OR        T0853	// R_OUT BUFFER DIE LD/PP SN ALARM
OUT       M00915	// R_OUT BUFFER DIE LD/PP SN ALARM
// =========================================================
// 
//       COUNT ALARM
// 
// =========================================================
; L622
LOAD      M00520
OUT       M00920
; L623
LOAD      M00521
OUT       M00921
; L624
LOAD      M00522
OUT       M00922
; L625
LOAD      M00523
OUT       M00923
; L626
LOAD      M00524
OUT       M00924
; L627
LOAD      M00525
OUT       M00925
; L628
LOAD      M00526
OUT       M00926
; L629
LOAD      M00527
OUT       M00927

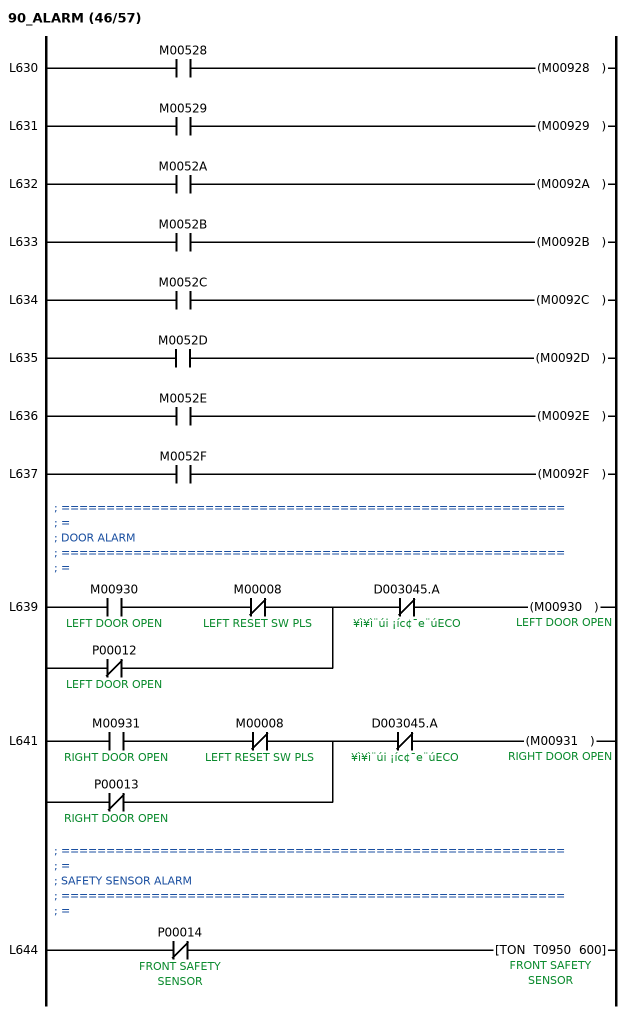
; L630
LOAD      M00528
OUT       M00928
; L631
LOAD      M00529
OUT       M00929
; L632
LOAD      M0052A
OUT       M0092A
; L633
LOAD      M0052B
OUT       M0092B
; L634
LOAD      M0052C
OUT       M0092C
; L635
LOAD      M0052D
OUT       M0092D
; L636
LOAD      M0052E
OUT       M0092E
; L637
LOAD      M0052F
OUT       M0092F
// =========================================================
// 
//       DOOR ALARM
// 
// =========================================================
; L639
LOAD      M00930	// LEFT DOOR OPEN
AND NOT   M00008	// LEFT RESET SW PLS
OR NOT    P00012	// LEFT DOOR OPEN
AND NOT   D003045.A	// ¥ì¥ì¨úi ¡íc¢¯e¨úECO
OUT       M00930	// LEFT DOOR OPEN
; L641
LOAD      M00931	// RIGHT DOOR OPEN
AND NOT   M00008	// LEFT RESET SW PLS
OR NOT    P00013	// RIGHT DOOR OPEN
AND NOT   D003045.A	// ¥ì¥ì¨úi ¡íc¢¯e¨úECO
OUT       M00931	// RIGHT DOOR OPEN
// =========================================================
// 
//       SAFETY SENSOR ALARM
// 
// =========================================================
; L644
LOAD NOT  P00014	// FRONT SAFETY SENSOR
TON       T0950 600	// FRONT SAFETY SENSOR

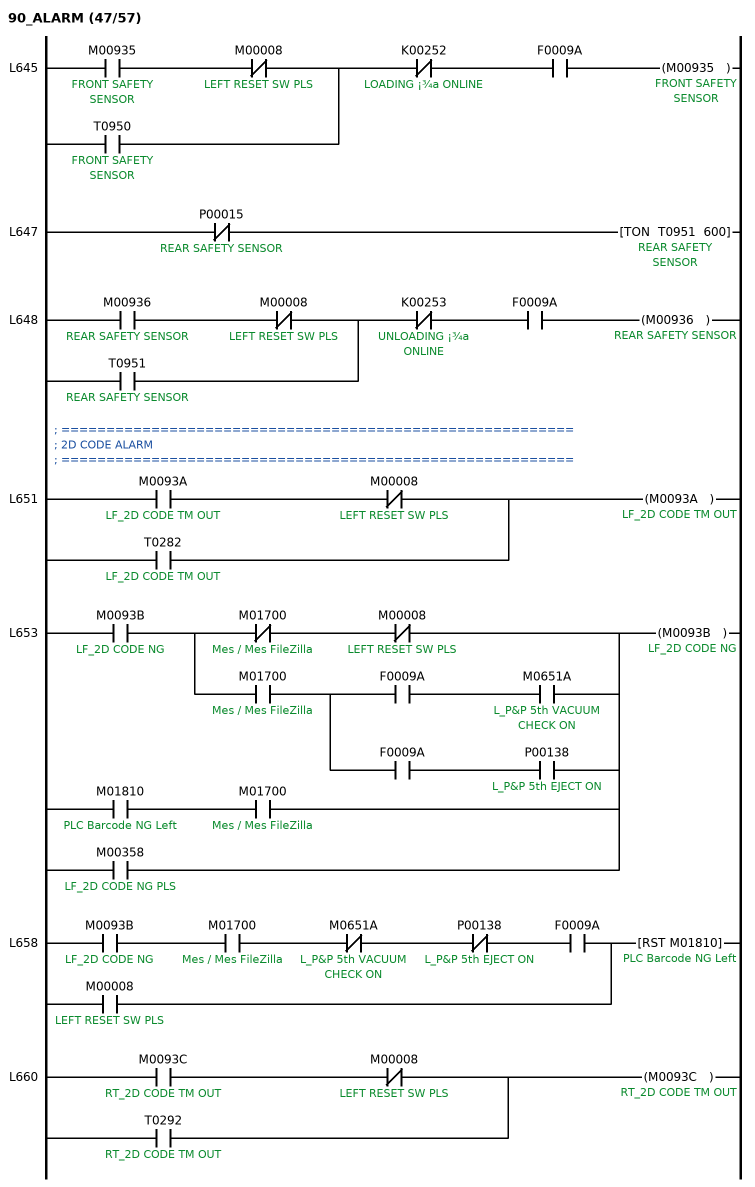
; L645
LOAD      M00935	// FRONT SAFETY SENSOR
AND NOT   M00008	// LEFT RESET SW PLS
OR        T0950	// FRONT SAFETY SENSOR
AND NOT   K00252	// LOADING ¡¾a ONLINE
AND       F0009A
OUT       M00935	// FRONT SAFETY SENSOR
; L647
LOAD NOT  P00015	// REAR SAFETY SENSOR
TON       T0951 600	// REAR SAFETY SENSOR
; L648
LOAD      M00936	// REAR SAFETY SENSOR
AND NOT   M00008	// LEFT RESET SW PLS
OR        T0951	// REAR SAFETY SENSOR
AND NOT   K00253	// UNLOADING ¡¾a ONLINE
AND       F0009A
OUT       M00936	// REAR SAFETY SENSOR
// =========================================================
// 
//       2D CODE ALARM
// 
// =========================================================
; L651
LOAD      M0093A	// LF_2D CODE TM OUT
AND NOT   M00008	// LEFT RESET SW PLS
OR        T0282	// LF_2D CODE TM OUT
OUT       M0093A	// LF_2D CODE TM OUT
; L653
LOAD      M0093B	// LF_2D CODE NG
LOAD NOT  M01700	// Mes / Mes FileZilla
AND NOT   M00008	// LEFT RESET SW PLS
LOAD      M01700	// Mes / Mes FileZilla
LOAD      F0009A
AND       M0651A	// L_P&P 5th VACUUM CHECK ON
LOAD      F0009A
AND       P00138	// L_P&P 5th EJECT ON
OR LOAD
AND LOAD
OR LOAD
AND LOAD
LOAD      M01810	// PLC Barcode NG Left
AND       M01700	// Mes / Mes FileZilla
OR LOAD
OR        M00358	// LF_2D CODE NG PLS
OUT       M0093B	// LF_2D CODE NG
; L658
LOAD      M0093B	// LF_2D CODE NG
AND       M01700	// Mes / Mes FileZilla
AND NOT   M0651A	// L_P&P 5th VACUUM CHECK ON
AND NOT   P00138	// L_P&P 5th EJECT ON
AND       F0009A
OR        M00008	// LEFT RESET SW PLS
RST       M01810	// PLC Barcode NG Left
; L660
LOAD      M0093C	// RT_2D CODE TM OUT
AND NOT   M00008	// LEFT RESET SW PLS
OR        T0292	// RT_2D CODE TM OUT
OUT       M0093C	// RT_2D CODE TM OUT

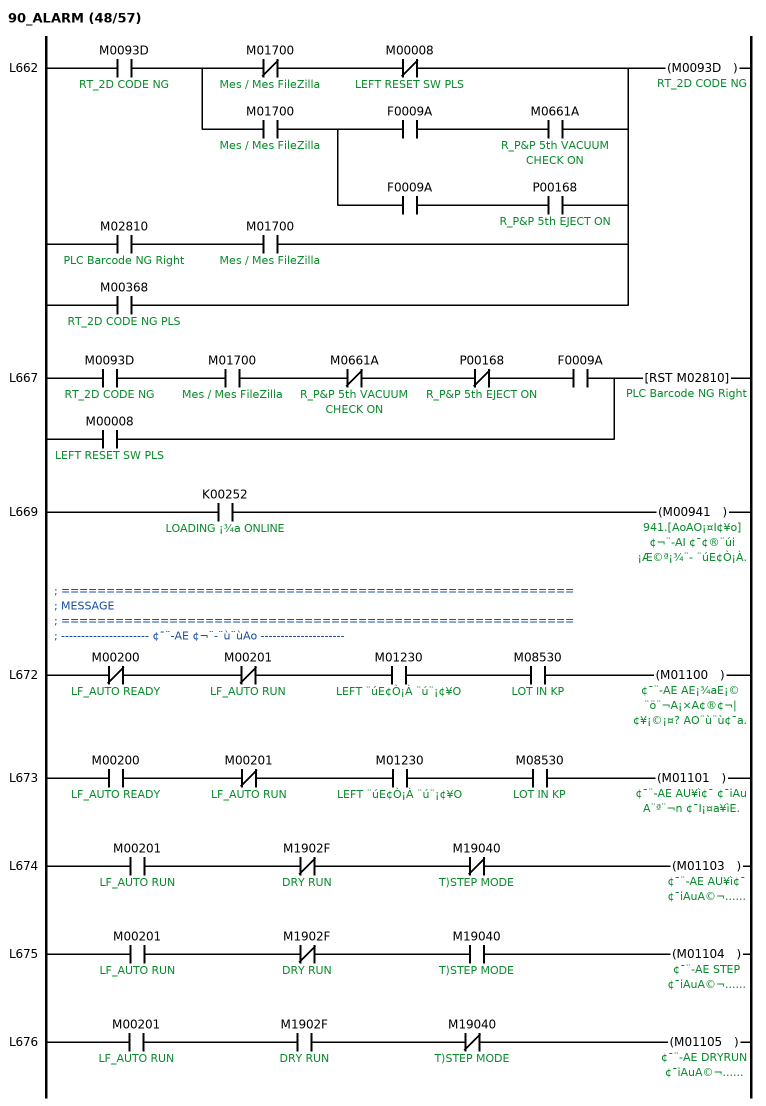
; L662
LOAD      M0093D	// RT_2D CODE NG
LOAD NOT  M01700	// Mes / Mes FileZilla
AND NOT   M00008	// LEFT RESET SW PLS
LOAD      M01700	// Mes / Mes FileZilla
LOAD      F0009A
AND       M0661A	// R_P&P 5th VACUUM CHECK ON
LOAD      F0009A
AND       P00168	// R_P&P 5th EJECT ON
OR LOAD
AND LOAD
OR LOAD
AND LOAD
LOAD      M02810	// PLC Barcode NG Right
AND       M01700	// Mes / Mes FileZilla
OR LOAD
OR        M00368	// RT_2D CODE NG PLS
OUT       M0093D	// RT_2D CODE NG
; L667
LOAD      M0093D	// RT_2D CODE NG
AND       M01700	// Mes / Mes FileZilla
AND NOT   M0661A	// R_P&P 5th VACUUM CHECK ON
AND NOT   P00168	// R_P&P 5th EJECT ON
AND       F0009A
OR        M00008	// LEFT RESET SW PLS
RST       M02810	// PLC Barcode NG Right
; L669
LOAD      K00252	// LOADING ¡¾a ONLINE
OUT       M00941	// 941.[AoAO¡¤I¢¥o] ¢¬¨­AI ¢¯¢®¨úi ¡Æ©ª¡¾¨­ ¨úE¢Ò¡À.
// =========================================================
// 
//       MESSAGE
// 
// =========================================================
// ---------------------- ¢¯¨­AE ¢¬¨­¨ù¨ùAo ---------------------
; L672
LOAD NOT  M00200	// LF_AUTO READY
AND NOT   M00201	// LF_AUTO RUN
AND       M01230	// LEFT ¨úE¢Ò¡À ¨ú¨¡¢¥O
AND       M08530	// LOT IN KP
OUT       M01100	// ¢¯¨­AE AE¡¾aE¡© ¨ö¨¬A¡×A¢®¢¬| ¢¥¡©¡¤? AO¨ù¨ù¢¯a.
; L673
LOAD      M00200	// LF_AUTO READY
AND NOT   M00201	// LF_AUTO RUN
AND       M01230	// LEFT ¨úE¢Ò¡À ¨ú¨¡¢¥O
AND       M08530	// LOT IN KP
OUT       M01101	// ¢¯¨­AE AU¥ì¢¯ ¢¯iAu A¨ª¨¬n ¢¯I¡¤a¥ìE.
; L674
LOAD      M00201	// LF_AUTO RUN
AND NOT   M1902F	// DRY RUN
AND NOT   M19040	// T)STEP MODE
OUT       M01103	// ¢¯¨­AE AU¥ì¢¯ ¢¯iAuA©¬......
; L675
LOAD      M00201	// LF_AUTO RUN
AND NOT   M1902F	// DRY RUN
AND       M19040	// T)STEP MODE
OUT       M01104	// ¢¯¨­AE STEP ¢¯iAuA©¬......
; L676
LOAD      M00201	// LF_AUTO RUN
AND       M1902F	// DRY RUN
AND NOT   M19040	// T)STEP MODE
OUT       M01105	// ¢¯¨­AE DRYRUN ¢¯iAuA©¬......

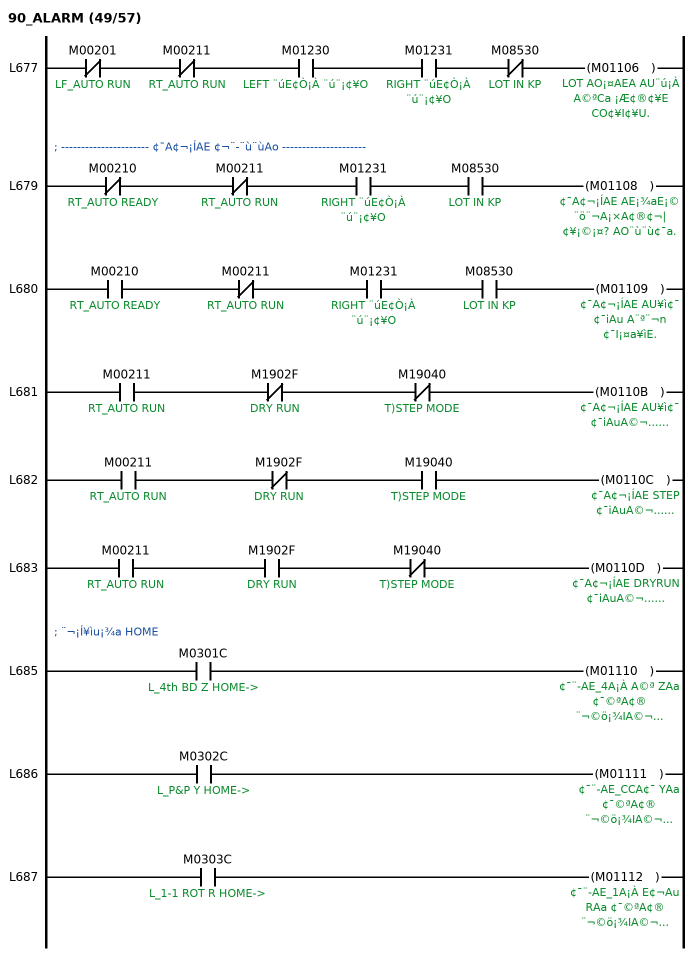
; L677
LOAD NOT  M00201	// LF_AUTO RUN
AND NOT   M00211	// RT_AUTO RUN
AND       M01230	// LEFT ¨úE¢Ò¡À ¨ú¨¡¢¥O
AND       M01231	// RIGHT ¨úE¢Ò¡À ¨ú¨¡¢¥O
AND NOT   M08530	// LOT IN KP
OUT       M01106	// LOT AO¡¤AEA AU¨ú¡À A©ªCa ¡Æ¢®¢¥E CO¢¥I¢¥U.
// ---------------------- ¢¯A¢¬¡ÍAE ¢¬¨­¨ù¨ùAo ---------------------
; L679
LOAD NOT  M00210	// RT_AUTO READY
AND NOT   M00211	// RT_AUTO RUN
AND       M01231	// RIGHT ¨úE¢Ò¡À ¨ú¨¡¢¥O
AND       M08530	// LOT IN KP
OUT       M01108	// ¢¯A¢¬¡ÍAE AE¡¾aE¡© ¨ö¨¬A¡×A¢®¢¬| ¢¥¡©¡¤? AO¨ù¨ù¢¯a.
; L680
LOAD      M00210	// RT_AUTO READY
AND NOT   M00211	// RT_AUTO RUN
AND       M01231	// RIGHT ¨úE¢Ò¡À ¨ú¨¡¢¥O
AND       M08530	// LOT IN KP
OUT       M01109	// ¢¯A¢¬¡ÍAE AU¥ì¢¯ ¢¯iAu A¨ª¨¬n ¢¯I¡¤a¥ìE.
; L681
LOAD      M00211	// RT_AUTO RUN
AND NOT   M1902F	// DRY RUN
AND NOT   M19040	// T)STEP MODE
OUT       M0110B	// ¢¯A¢¬¡ÍAE AU¥ì¢¯ ¢¯iAuA©¬......
; L682
LOAD      M00211	// RT_AUTO RUN
AND NOT   M1902F	// DRY RUN
AND       M19040	// T)STEP MODE
OUT       M0110C	// ¢¯A¢¬¡ÍAE STEP ¢¯iAuA©¬......
; L683
LOAD      M00211	// RT_AUTO RUN
AND       M1902F	// DRY RUN
AND NOT   M19040	// T)STEP MODE
OUT       M0110D	// ¢¯A¢¬¡ÍAE DRYRUN ¢¯iAuA©¬......
// ¨¬¡Í¥ìu¡¾a HOME
; L685
LOAD      M0301C	// L_4th BD Z HOME->
OUT       M01110	// ¢¯¨­AE_4A¡À A©ª ZAa ¢¯©ªA¢® ¨¬©ö¡¾IA©¬...
; L686
LOAD      M0302C	// L_P&P Y HOME->
OUT       M01111	// ¢¯¨­AE_CCA¢¯ YAa ¢¯©ªA¢® ¨¬©ö¡¾IA©¬...
; L687
LOAD      M0303C	// L_1-1 ROT R HOME->
OUT       M01112	// ¢¯¨­AE_1A¡À E¢¬Au RAa ¢¯©ªA¢® ¨¬©ö¡¾IA©¬...

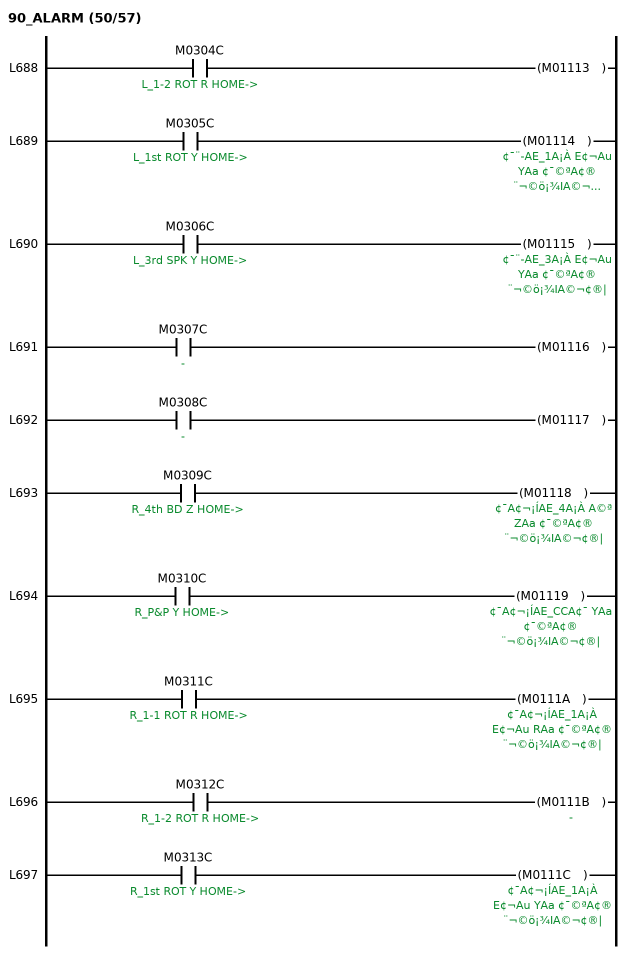
; L688
LOAD      M0304C	// L_1-2 ROT R HOME->
OUT       M01113
; L689
LOAD      M0305C	// L_1st ROT Y HOME->
OUT       M01114	// ¢¯¨­AE_1A¡À E¢¬Au YAa ¢¯©ªA¢® ¨¬©ö¡¾IA©¬...
; L690
LOAD      M0306C	// L_3rd SPK Y HOME->
OUT       M01115	// ¢¯¨­AE_3A¡À E¢¬Au YAa ¢¯©ªA¢® ¨¬©ö¡¾IA©¬¢®|
; L691
LOAD      M0307C	// -
OUT       M01116
; L692
LOAD      M0308C	// -
OUT       M01117
; L693
LOAD      M0309C	// R_4th BD Z HOME->
OUT       M01118	// ¢¯A¢¬¡ÍAE_4A¡À A©ª ZAa ¢¯©ªA¢® ¨¬©ö¡¾IA©¬¢®|
; L694
LOAD      M0310C	// R_P&P Y HOME->
OUT       M01119	// ¢¯A¢¬¡ÍAE_CCA¢¯ YAa ¢¯©ªA¢® ¨¬©ö¡¾IA©¬¢®|
; L695
LOAD      M0311C	// R_1-1 ROT R HOME->
OUT       M0111A	// ¢¯A¢¬¡ÍAE_1A¡À E¢¬Au RAa ¢¯©ªA¢® ¨¬©ö¡¾IA©¬¢®|
; L696
LOAD      M0312C	// R_1-2 ROT R HOME->
OUT       M0111B	// -
; L697
LOAD      M0313C	// R_1st ROT Y HOME->
OUT       M0111C	// ¢¯A¢¬¡ÍAE_1A¡À E¢¬Au YAa ¢¯©ªA¢® ¨¬©ö¡¾IA©¬¢®|

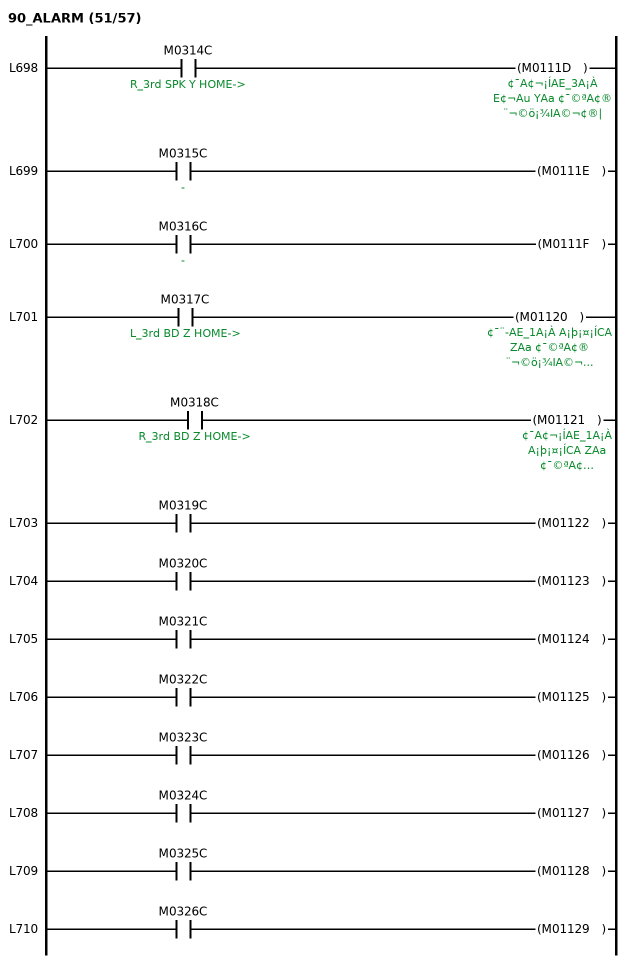
; L698
LOAD      M0314C	// R_3rd SPK Y HOME->
OUT       M0111D	// ¢¯A¢¬¡ÍAE_3A¡À E¢¬Au YAa ¢¯©ªA¢® ¨¬©ö¡¾IA©¬¢®|
; L699
LOAD      M0315C	// -
OUT       M0111E
; L700
LOAD      M0316C	// -
OUT       M0111F
; L701
LOAD      M0317C	// L_3rd BD Z HOME->
OUT       M01120	// ¢¯¨­AE_1A¡À A¡þ¡¤¡ÍCA ZAa ¢¯©ªA¢® ¨¬©ö¡¾IA©¬...
; L702
LOAD      M0318C	// R_3rd BD Z HOME->
OUT       M01121	// ¢¯A¢¬¡ÍAE_1A¡À A¡þ¡¤¡ÍCA ZAa ¢¯©ªA¢® ¨¬©ö¡¾IA©¬...
; L703
LOAD      M0319C
OUT       M01122
; L704
LOAD      M0320C
OUT       M01123
; L705
LOAD      M0321C
OUT       M01124
; L706
LOAD      M0322C
OUT       M01125
; L707
LOAD      M0323C
OUT       M01126
; L708
LOAD      M0324C
OUT       M01127
; L709
LOAD      M0325C
OUT       M01128
; L710
LOAD      M0326C
OUT       M01129

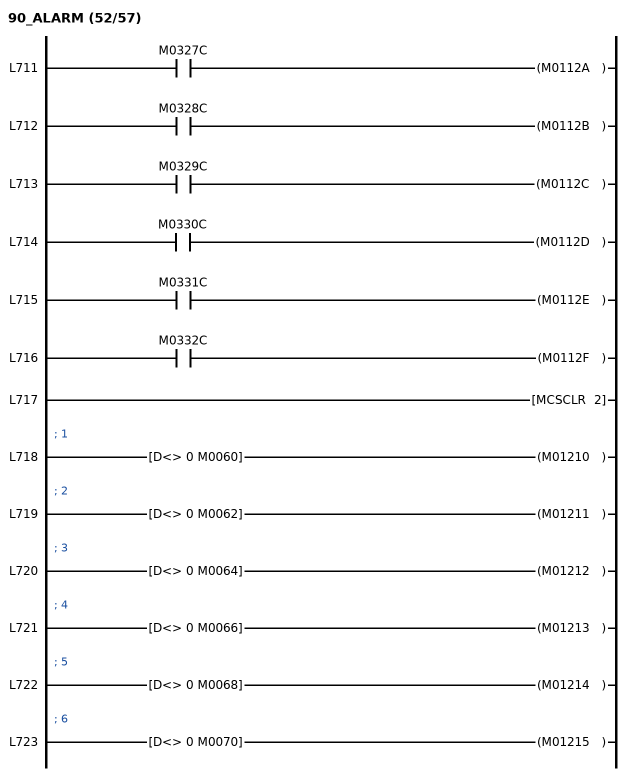
; L711
LOAD      M0327C
OUT       M0112A
; L712
LOAD      M0328C
OUT       M0112B
; L713
LOAD      M0329C
OUT       M0112C
; L714
LOAD      M0330C
OUT       M0112D
; L715
LOAD      M0331C
OUT       M0112E
; L716
LOAD      M0332C
OUT       M0112F
; L717
MCSCLR    2
; L718
LOADD<>   0 M0060
OUT       M01210
// output comment: 1
; L719
LOADD<>   0 M0062
OUT       M01211
// output comment: 2
; L720
LOADD<>   0 M0064
OUT       M01212
// output comment: 3
; L721
LOADD<>   0 M0066
OUT       M01213
// output comment: 4
; L722
LOADD<>   0 M0068
OUT       M01214
// output comment: 5
; L723
LOADD<>   0 M0070
OUT       M01215
// output comment: 6

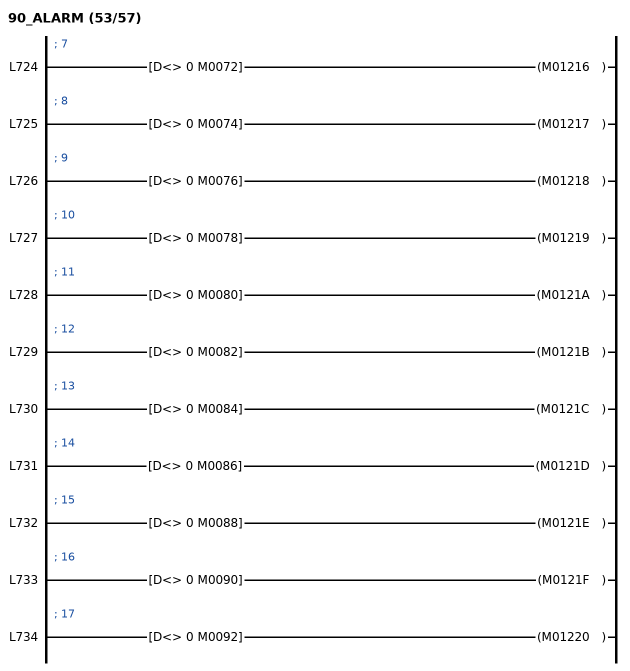
; L724
LOADD<>   0 M0072
OUT       M01216
// output comment: 7
; L725
LOADD<>   0 M0074
OUT       M01217
// output comment: 8
; L726
LOADD<>   0 M0076
OUT       M01218
// output comment: 9
; L727
LOADD<>   0 M0078
OUT       M01219
// output comment: 10
; L728
LOADD<>   0 M0080
OUT       M0121A
// output comment: 11
; L729
LOADD<>   0 M0082
OUT       M0121B
// output comment: 12
; L730
LOADD<>   0 M0084
OUT       M0121C
// output comment: 13
; L731
LOADD<>   0 M0086
OUT       M0121D
// output comment: 14
; L732
LOADD<>   0 M0088
OUT       M0121E
// output comment: 15
; L733
LOADD<>   0 M0090
OUT       M0121F
// output comment: 16
; L734
LOADD<>   0 M0092
OUT       M01220
// output comment: 17

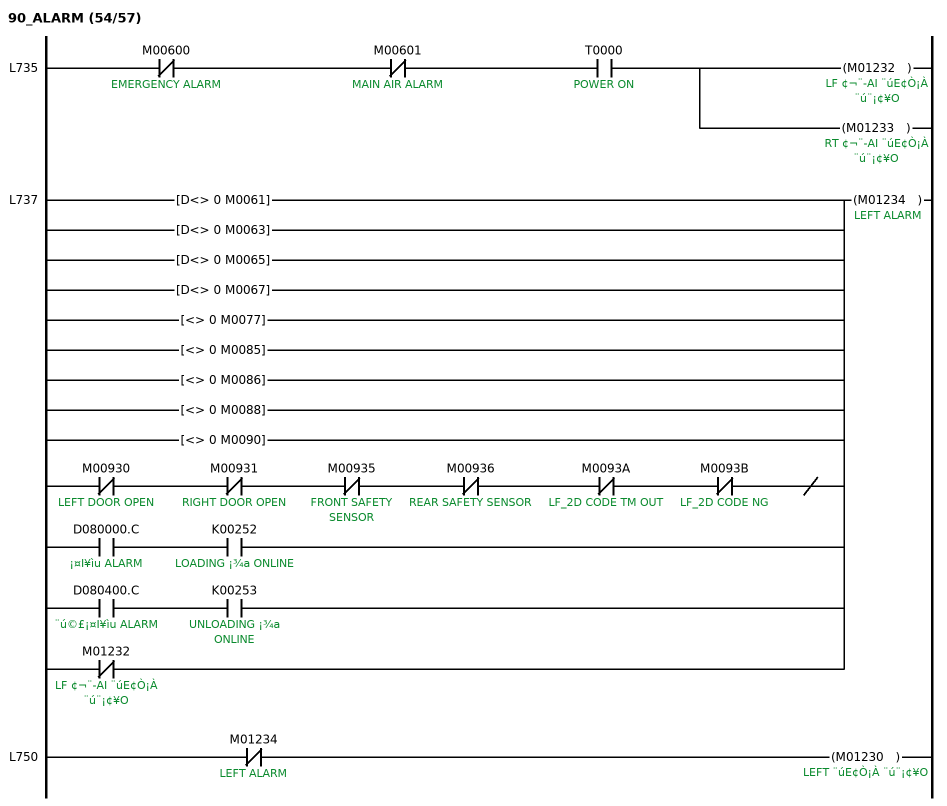
; L735
LOAD NOT  M00600	// EMERGENCY ALARM
AND NOT   M00601	// MAIN AIR ALARM
AND       T0000	// POWER ON
OUT       M01232	// LF ¢¬¨­AI ¨úE¢Ò¡À ¨ú¨¡¢¥O
OUT       M01233	// RT ¢¬¨­AI ¨úE¢Ò¡À ¨ú¨¡¢¥O
; L737
LOADD<>   0 M0061
ORD<>     0 M0063
ORD<>     0 M0065
ORD<>     0 M0067
OR<>      0 M0077
OR<>      0 M0085
OR<>      0 M0086
OR<>      0 M0088
OR<>      0 M0090
LOAD NOT  M00930	// LEFT DOOR OPEN
AND NOT   M00931	// RIGHT DOOR OPEN
AND NOT   M00935	// FRONT SAFETY SENSOR
AND NOT   M00936	// REAR SAFETY SENSOR
AND NOT   M0093A	// LF_2D CODE TM OUT
AND NOT   M0093B	// LF_2D CODE NG
NOT
OR LOAD
LOAD      D080000.C	// ¡¤I¥ìu ALARM
AND       K00252	// LOADING ¡¾a ONLINE
OR LOAD
LOAD      D080400.C	// ¨ú©£¡¤I¥ìu ALARM
AND       K00253	// UNLOADING ¡¾a ONLINE
OR LOAD
OR NOT    M01232	// LF ¢¬¨­AI ¨úE¢Ò¡À ¨ú¨¡¢¥O
OUT       M01234	// LEFT ALARM
; L750
LOAD NOT  M01234	// LEFT ALARM
OUT       M01230	// LEFT ¨úE¢Ò¡À ¨ú¨¡¢¥O

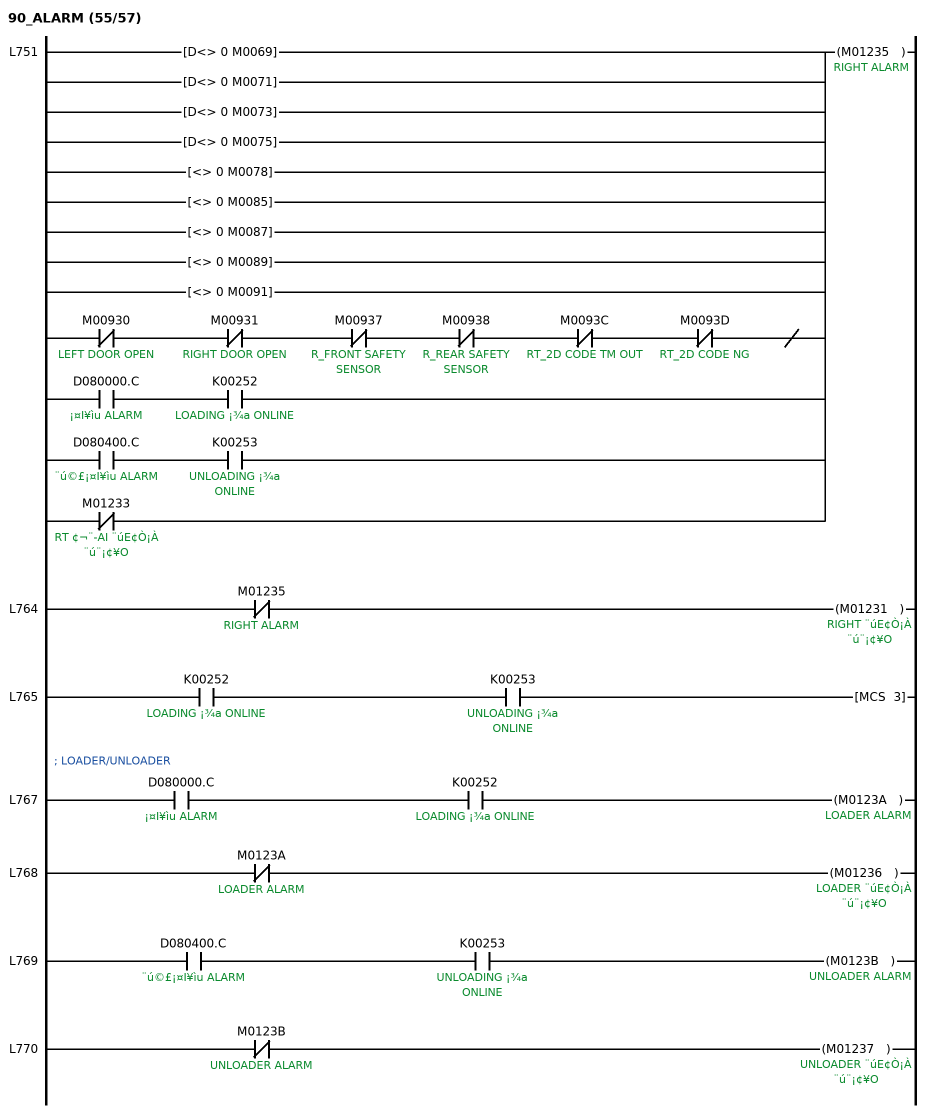
; L751
LOADD<>   0 M0069
ORD<>     0 M0071
ORD<>     0 M0073
ORD<>     0 M0075
OR<>      0 M0078
OR<>      0 M0085
OR<>      0 M0087
OR<>      0 M0089
OR<>      0 M0091
LOAD NOT  M00930	// LEFT DOOR OPEN
AND NOT   M00931	// RIGHT DOOR OPEN
AND NOT   M00937	// R_FRONT SAFETY SENSOR
AND NOT   M00938	// R_REAR SAFETY SENSOR
AND NOT   M0093C	// RT_2D CODE TM OUT
AND NOT   M0093D	// RT_2D CODE NG
NOT
OR LOAD
LOAD      D080000.C	// ¡¤I¥ìu ALARM
AND       K00252	// LOADING ¡¾a ONLINE
OR LOAD
LOAD      D080400.C	// ¨ú©£¡¤I¥ìu ALARM
AND       K00253	// UNLOADING ¡¾a ONLINE
OR LOAD
OR NOT    M01233	// RT ¢¬¨­AI ¨úE¢Ò¡À ¨ú¨¡¢¥O
OUT       M01235	// RIGHT ALARM
; L764
LOAD NOT  M01235	// RIGHT ALARM
OUT       M01231	// RIGHT ¨úE¢Ò¡À ¨ú¨¡¢¥O
; L765
LOAD      K00252	// LOADING ¡¾a ONLINE
AND       K00253	// UNLOADING ¡¾a ONLINE
MCS       3
// LOADER/UNLOADER
; L767
LOAD      D080000.C	// ¡¤I¥ìu ALARM
AND       K00252	// LOADING ¡¾a ONLINE
OUT       M0123A	// LOADER ALARM
; L768
LOAD NOT  M0123A	// LOADER ALARM
OUT       M01236	// LOADER ¨úE¢Ò¡À ¨ú¨¡¢¥O
; L769
LOAD      D080400.C	// ¨ú©£¡¤I¥ìu ALARM
AND       K00253	// UNLOADING ¡¾a ONLINE
OUT       M0123B	// UNLOADER ALARM
; L770
LOAD NOT  M0123B	// UNLOADER ALARM
OUT       M01237	// UNLOADER ¨úE¢Ò¡À ¨ú¨¡¢¥O

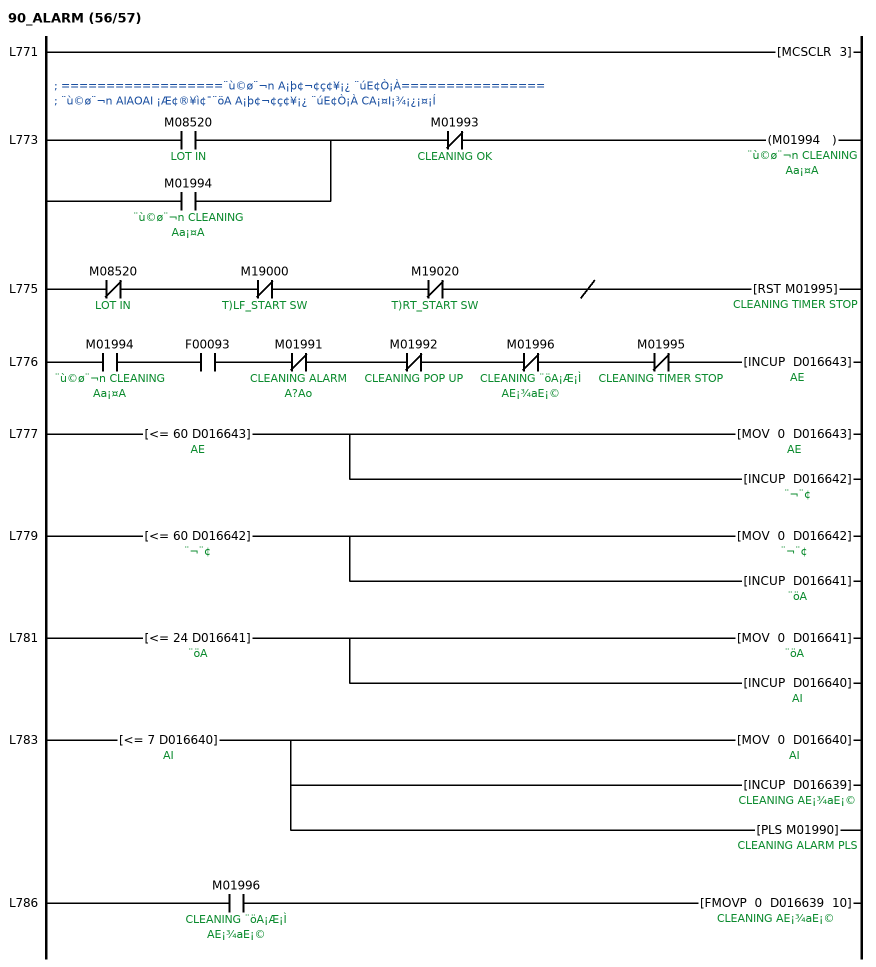
; L771
MCSCLR    3
// ==================¨ù©ø¨¬n A¡þ¢¬¢ç¢¥¡¿ ¨úE¢Ò¡À================
; L773
LOAD      M08520	// LOT IN
OR        M01994	// ¨ù©ø¨¬n CLEANING Aa¡¤A
AND NOT   M01993	// CLEANING OK
OUT       M01994	// ¨ù©ø¨¬n CLEANING Aa¡¤A
// output comment: ¨ù©ø¨¬n AIAOAI ¡Æ¢®¥ì¢¯¨öA A¡þ¢¬¢ç¢¥¡¿ ¨úE¢Ò¡À CA¡¤I¡¾¡¿¡¤¡Í
; L775
LOAD NOT  M08520	// LOT IN
AND NOT   M19000	// T)LF_START SW
AND NOT   M19020	// T)RT_START SW
NOT
RST       M01995	// CLEANING TIMER STOP
; L776
LOAD      M01994	// ¨ù©ø¨¬n CLEANING Aa¡¤A
AND       F00093
AND NOT   M01991	// CLEANING ALARM A?Ao
AND NOT   M01992	// CLEANING POP UP
AND NOT   M01996	// CLEANING ¨öA¡Æ¡Ì AE¡¾aE¡©
AND NOT   M01995	// CLEANING TIMER STOP
INCUP     D016643	// AE
; L777
LOAD<=    60 D016643	// AE
MOV       0 D016643	// AE
INCUP     D016642	// ¨¬¨¢
; L779
LOAD<=    60 D016642	// ¨¬¨¢
MOV       0 D016642	// ¨¬¨¢
INCUP     D016641	// ¨öA
; L781
LOAD<=    24 D016641	// ¨öA
MOV       0 D016641	// ¨öA
INCUP     D016640	// AI
; L783
LOAD<=    7 D016640	// AI
MOV       0 D016640	// AI
INCUP     D016639	// CLEANING AE¡¾aE¡©
OUTP      M01990	// CLEANING ALARM PLS
; L786
LOAD      M01996	// CLEANING ¨öA¡Æ¡Ì AE¡¾aE¡©
FMOVP     0 D016639 10	// CLEANING AE¡¾aE¡©

